LIN {X 0,Y 122.417,Z 271.708,A -85,B 0,C 180,E1 -25566.608,E2 -25566.608} C_VEL
LIN {X 0,Y 122.316,Z 271.702,A -85,B 0,C 180,E1 -25572.377,E2 -25572.377} C_VEL
LIN {X 0,Y 122.102,Z 271.77,A -85,B 0,C 180,E1 -25576.74,E2 -25576.74} C_VEL
LIN {X 0,Y 122.036,Z 271.748,A -85,B 0,C 180,E1 -25582.868,E2 -25582.868} C_VEL
LIN {X 0,Y 121.951,Z 271.777,A -85,B 0,C 180,E1 -25587.47,E2 -25587.47} C_VEL
LIN {X 0,Y 121.974,Z 272.027,A -85,B 0,C 180,E1 -25592.04,E2 -25592.04} C_VEL
LIN {X 0,Y 122.267,Z 273.161,A -85,B 0,C 180,E1 -25592.746,E2 -25592.746} C_VEL
LIN {X 0,Y 123.853,Z 275.808,A -85,B 0,C 180,E1 -25593.851,E2 -25593.851} C_VEL
LIN {X 0,Y 125.36,Z 277.295,A -85,B 0,C 180,E1 -25594.741,E2 -25594.741} C_VEL
LIN {X 0,Y 127.561,Z 280.725,A -85,B 0,C 180,E1 -25596.09,E2 -25596.09} C_VEL
LIN {X 0,Y 133.318,Z 289.437,A -85,B 0,C 180,E1 -25599.257,E2 -25599.257} C_VEL
LIN {X 0,Y 139.122,Z 299.64,A -85,B 0,C 180,E1 -25602.154,E2 -25602.154} C_VEL
LIN {X 0,Y 143.343,Z 310.259,A -85,B 0,C 180,E1 -25604.257,E2 -25604.257} C_VEL
LIN {X 0,Y 147.015,Z 321.622,A -85,B 0,C 180,E1 -25606.074,E2 -25606.074} C_VEL
LIN {X 0,Y 147.266,Z 325.906,A -85,B 0,C 180,E1 -25606.408,E2 -25606.408} C_VEL
LIN {X 0,Y 144.065,Z 374.094,A -85,B 0,C 180,E1 -25608.57,E2 -25608.57} C_VEL
LIN {X 0,Y 142.298,Z 387.376,A -85,B 0,C 180,E1 -25609.638,E2 -25609.638} C_VEL
LIN {X 0,Y 140.096,Z 399.712,A -85,B 0,C 180,E1 -25611.167,E2 -25611.167} C_VEL
LIN {X 0,Y 137.398,Z 410.903,A -85,B 0,C 180,E1 -25613.058,E2 -25613.058} C_VEL
LIN {X 0,Y 134.822,Z 419.925,A -85,B 0,C 180,E1 -25615.013,E2 -25615.013} C_VEL
LIN {X 0,Y 131.525,Z 430.91,A -85,B 0,C 180,E1 -25618.154,E2 -25618.154} C_VEL
LIN {X 0,Y 128.19,Z 440.642,A -85,B 0,C 180,E1 -25621.736,E2 -25621.736} C_VEL
LIN {X 0,Y 125.67,Z 448.029,A -85,B 0,C 180,E1 -25625.203,E2 -25625.203} C_VEL
LIN {X 0,Y 122.916,Z 456.04,A -85,B 0,C 180,E1 -25629.938,E2 -25629.938} C_VEL
LIN {X 0,Y 121.019,Z 462.413,A -85,B 0,C 180,E1 -25634.852,E2 -25634.852} C_VEL
LIN {X 0,Y 119.82,Z 467.456,A -85,B 0,C 180,E1 -25639.866,E2 -25639.866} C_VEL
LIN {X 0,Y 119.27,Z 471.332,A -85,B 0,C 180,E1 -25644.93,E2 -25644.93} C_VEL
LIN {X 0,Y 119.304,Z 474.157,A -85,B 0,C 180,E1 -25650.001,E2 -25650.001} C_VEL
LIN {X 0,Y 119.247,Z 475.469,A -85,B 0,C 180,E1 -25653.38,E2 -25653.38} C_VEL
LIN {X 0,Y 119.98,Z 476.932,A -85,B 0,C 180,E1 -25660.122,E2 -25660.122} C_VEL
LIN {X 0,Y 121.968,Z 476.809,A -85,B 0,C 180,E1 -25666.691,E2 -25666.691} C_VEL
LIN {X 0,Y 125.493,Z 475.157,A -85,B 0,C 180,E1 -25673.081,E2 -25673.081} C_VEL
LIN {X 0,Y 127.894,Z 473.752,A -85,B 0,C 180,E1 -25676.08,E2 -25676.08} C_VEL
LIN {X 0,Y 131.395,Z 471.343,A -85,B 0,C 180,E1 -25679.691,E2 -25679.691} C_VEL
LIN {X 0,Y 133.223,Z 469.569,A -85,B 0,C 180,E1 -25682.001,E2 -25682.001} C_VEL
LIN {X 0,Y 134.965,Z 466.294,A -85,B 0,C 180,E1 -25685.937,E2 -25685.937} C_VEL
LIN {X 0,Y 137.186,Z 462.408,A -85,B 0,C 180,E1 -25689.659,E2 -25689.659} C_VEL
LIN {X 0,Y 139.665,Z 459.633,A -85,B 0,C 180,E1 -25691.56,E2 -25691.56} C_VEL
LIN {X 0,Y 146.623,Z 452.507,A -85,B 0,C 180,E1 -25694.993,E2 -25694.993} C_VEL
LIN {X 0,Y 153.812,Z 443.935,A -85,B 0,C 180,E1 -25697.946,E2 -25697.946} C_VEL
LIN {X 0,Y 160.067,Z 435.206,A -85,B 0,C 180,E1 -25700.208,E2 -25700.208} C_VEL
LIN {X 0,Y 165.907,Z 425.657,A -85,B 0,C 180,E1 -25702.091,E2 -25702.091} C_VEL
LIN {X 0,Y 171.308,Z 415.227,A -85,B 0,C 180,E1 -25703.624,E2 -25703.624} C_VEL
LIN {X 0,Y 176.137,Z 403.695,A -85,B 0,C 180,E1 -25704.883,E2 -25704.883} C_VEL
LIN {X 0,Y 180.007,Z 391.632,A -85,B 0,C 180,E1 -25705.852,E2 -25705.852} C_VEL
LIN {X 0,Y 183.062,Z 378.393,A -85,B 0,C 180,E1 -25706.585,E2 -25706.585} C_VEL
LIN {X 0,Y 184.796,Z 365.742,A -85,B 0,C 180,E1 -25707.042,E2 -25707.042} C_VEL
LIN {X 0,Y 185.317,Z 359.615,A -85,B 0,C 180,E1 -25707.264,E2 -25707.264} C_VEL
LIN {X 0,Y 182.402,Z 351.71,A -85,B 0,C 180,E1 -25710.159,E2 -25710.159} C_VEL
LIN {X 0,Y 179.342,Z 344.498,A -85,B 0,C 180,E1 -25713.644,E2 -25713.644} C_VEL
LIN {X 0,Y 177.139,Z 339.924,A -85,B 0,C 180,E1 -25716.615,E2 -25716.615} C_VEL
LIN {X 0,Y 175.755,Z 337.207,A -85,B 0,C 180,E1 -25718.897,E2 -25718.897} C_VEL
LIN {X 0,Y 173.712,Z 333.275,A -85,B 0,C 180,E1 -25723.538,E2 -25723.538} C_VEL
LIN {X 0,Y 172.304,Z 331.593,A -85,B 0,C 180,E1 -25730.6,E2 -25730.6} C_VEL
LIN {X 0,Y 173.403,Z 332.544,A -85,B 0,C 180,E1 -25737.667,E2 -25737.667} C_VEL
LIN {X 0,Y 173.905,Z 333.209,A -85,B 0,C 180,E1 -25739.121,E2 -25739.121} C_VEL
LIN {X 0,Y 175.898,Z 336.978,A -85,B 0,C 180,E1 -25743.5,E2 -25743.5} C_VEL
LIN {X 0,Y 178.522,Z 341.814,A -85,B 0,C 180,E1 -25747.418,E2 -25747.418} C_VEL
LIN {X 0,Y 180.756,Z 345.931,A -85,B 0,C 180,E1 -25750.065,E2 -25750.065} C_VEL
LIN {X 0,Y 182.611,Z 349.737,A -85,B 0,C 180,E1 -25752.028,E2 -25752.028} C_VEL
LIN {X 0,Y 185.533,Z 357.045,A -85,B 0,C 180,E1 -25754.874,E2 -25754.874} C_VEL
LIN {X 0,Y 183.565,Z 374.418,A -85,B 0,C 180,E1 -25755.499,E2 -25755.499} C_VEL
LIN {X 0,Y 180.942,Z 386.69,A -85,B 0,C 180,E1 -25756.119,E2 -25756.119} C_VEL
LIN {X 0,Y 177.256,Z 398.948,A -85,B 0,C 180,E1 -25757.071,E2 -25757.071} C_VEL
LIN {X 0,Y 172.252,Z 411.617,A -85,B 0,C 180,E1 -25758.446,E2 -25758.446} C_VEL
LIN {X 0,Y 167.111,Z 421.976,A -85,B 0,C 180,E1 -25759.962,E2 -25759.962} C_VEL
LIN {X 0,Y 160.993,Z 432.133,A -85,B 0,C 180,E1 -25761.927,E2 -25761.927} C_VEL
LIN {X 0,Y 154.339,Z 441.539,A -85,B 0,C 180,E1 -25764.393,E2 -25764.393} C_VEL
LIN {X 0,Y 148,Z 449.237,A -85,B 0,C 180,E1 -25767.078,E2 -25767.078} C_VEL
LIN {X 0,Y 141.389,Z 456.166,A -85,B 0,C 180,E1 -25770.301,E2 -25770.301} C_VEL
LIN {X 0,Y 135.346,Z 461.683,A -85,B 0,C 180,E1 -25773.816,E2 -25773.816} C_VEL
LIN {X 0,Y 129.352,Z 466.403,A -85,B 0,C 180,E1 -25778.016,E2 -25778.016} C_VEL
LIN {X 0,Y 123.843,Z 470.088,A -85,B 0,C 180,E1 -25782.899,E2 -25782.899} C_VEL
LIN {X 0,Y 121.135,Z 471.63,A -85,B 0,C 180,E1 -25785.874,E2 -25785.874} C_VEL
LIN {X 0,Y 117.41,Z 473.328,A -85,B 0,C 180,E1 -25791.065,E2 -25791.065} C_VEL
LIN {X 0,Y 114.591,Z 474.002,A -85,B 0,C 180,E1 -25796.496,E2 -25796.496} C_VEL
LIN {X 0,Y 113.253,Z 473.913,A -85,B 0,C 180,E1 -25800.281,E2 -25800.281} C_VEL
LIN {X 0,Y 112.337,Z 473.353,A -85,B 0,C 180,E1 -25804.027,E2 -25804.027} C_VEL
LIN {X 0,Y 111.648,Z 471.307,A -85,B 0,C 180,E1 -25810.716,E2 -25810.716} C_VEL
LIN {X 0,Y 111.953,Z 467.915,A -85,B 0,C 180,E1 -25817.306,E2 -25817.306} C_VEL
LIN {X 0,Y 113.091,Z 463.049,A -85,B 0,C 180,E1 -25823.712,E2 -25823.712} C_VEL
LIN {X 0,Y 115.123,Z 456.472,A -85,B 0,C 180,E1 -25829.999,E2 -25829.999} C_VEL
LIN {X 0,Y 117.55,Z 449.355,A -85,B 0,C 180,E1 -25835.144,E2 -25835.144} C_VEL
LIN {X 0,Y 120.797,Z 440.409,A -85,B 0,C 180,E1 -25840.051,E2 -25840.051} C_VEL
LIN {X 0,Y 124.177,Z 431.212,A -85,B 0,C 180,E1 -25843.917,E2 -25843.917} C_VEL
LIN {X 0,Y 127.578,Z 421.06,A -85,B 0,C 180,E1 -25847.222,E2 -25847.222} C_VEL
LIN {X 0,Y 130.961,Z 409.719,A -85,B 0,C 180,E1 -25850.004,E2 -25850.004} C_VEL
LIN {X 0,Y 134.071,Z 397.023,A -85,B 0,C 180,E1 -25852.335,E2 -25852.335} C_VEL
LIN {X 0,Y 136.353,Z 384.7,A -85,B 0,C 180,E1 -25853.946,E2 -25853.946} C_VEL
LIN {X 0,Y 138.276,Z 370.597,A -85,B 0,C 180,E1 -25855.122,E2 -25855.122} C_VEL
LIN {X 0,Y 141.666,Z 320.771,A -85,B 0,C 180,E1 -25857.421,E2 -25857.421} C_VEL
LIN {X 0,Y 138.482,Z 311.486,A -85,B 0,C 180,E1 -25859.089,E2 -25859.089} C_VEL
LIN {X 0,Y 131.285,Z 297.708,A -85,B 0,C 180,E1 -25862.78,E2 -25862.78} C_VEL
LIN {X 0,Y 124.325,Z 286.522,A -85,B 0,C 180,E1 -25866.815,E2 -25866.815} C_VEL
LIN {X 0,Y 121.077,Z 282.094,A -85,B 0,C 180,E1 -25868.889,E2 -25868.889} C_VEL
LIN {X 0,Y 118.948,Z 279.166,A -85,B 0,C 180,E1 -25870.362,E2 -25870.362} C_VEL
LIN {X 0,Y 118.239,Z 277.828,A -85,B 0,C 180,E1 -25870.91,E2 -25870.91} C_VEL
LIN {X 0,Y 115.881,Z 275.514,A -85,B 0,C 180,E1 -25872.61,E2 -25872.61} C_VEL
LIN {X 0,Y 114.976,Z 273.193,A -85,B 0,C 180,E1 -25873.766,E2 -25873.766} C_VEL
LIN {X 0,Y 114.847,Z 272.682,A -85,B 0,C 180,E1 -25875.203,E2 -25875.203} C_VEL
LIN {X 0,Y 114.852,Z 272.662,A -85,B 0,C 180,E1 -25877.716,E2 -25877.716} C_VEL
LIN {X 0,Y 114.833,Z 272.637,A -85,B 0,C 180,E1 -25882.712,E2 -25882.712} C_VEL
LIN {X 0,Y 114.844,Z 272.645,A -85,B 0,C 180,E1 -25888.95,E2 -25888.95} C_VEL
LIN {X 0,Y 114.946,Z 272.645,A -85,B 0,C 180,E1 -25896.506,E2 -25896.506} C_VEL
LIN {X 0,Y 115.016,Z 272.604,A -85,B 0,C 180,E1 -25902.228,E2 -25902.228} C_VEL
LIN {X 0,Y 115.276,Z 272.57,A -85,B 0,C 180,E1 -25907.276,E2 -25907.276} C_VEL
LIN {X 0,Y 115.387,Z 272.593,A -85,B 0,C 180,E1 -25913.019,E2 -25913.019} C_VEL
LIN {X 0,Y 115.989,Z 272.479,A -85,B 0,C 180,E1 -25920.016,E2 -25920.016} C_VEL
LIN {X 0,Y 115.359,Z 272.578,A -85,B 0,C 180,E1 -25927.014,E2 -25927.014} C_VEL
LIN {X 0,Y 115.252,Z 272.583,A -85,B 0,C 180,E1 -25932.672,E2 -25932.672} C_VEL
LIN {X 0,Y 115.006,Z 272.635,A -85,B 0,C 180,E1 -25937.807,E2 -25937.807} C_VEL
LIN {X 0,Y 114.955,Z 272.635,A -85,B 0,C 180,E1 -25943.505,E2 -25943.505} C_VEL
LIN {X 0,Y 114.957,Z 272.956,A -85,B 0,C 180,E1 -25947.802,E2 -25947.802} C_VEL
LIN {X 0,Y 115.218,Z 274.115,A -85,B 0,C 180,E1 -25948.6,E2 -25948.6} C_VEL
LIN {X 0,Y 116.721,Z 276.593,A -85,B 0,C 180,E1 -25949.868,E2 -25949.868} C_VEL
LIN {X 0,Y 118.61,Z 278.382,A -85,B 0,C 180,E1 -25951.197,E2 -25951.197} C_VEL
LIN {X 0,Y 120.6,Z 281.579,A -85,B 0,C 180,E1 -25952.635,E2 -25952.635} C_VEL
LIN {X 0,Y 122.018,Z 283.329,A -85,B 0,C 180,E1 -25953.56,E2 -25953.56} C_VEL
LIN {X 0,Y 127.424,Z 291.559,A -85,B 0,C 180,E1 -25956.909,E2 -25956.909} C_VEL
LIN {X 0,Y 132.932,Z 300.828,A -85,B 0,C 180,E1 -25959.946,E2 -25959.946} C_VEL
LIN {X 0,Y 135.86,Z 307.143,A -85,B 0,C 180,E1 -25961.513,E2 -25961.513} C_VEL
LIN {X 0,Y 140.144,Z 319.557,A -85,B 0,C 180,E1 -25963.842,E2 -25963.842} C_VEL
LIN {X 0,Y 141.499,Z 323.985,A -85,B 0,C 180,E1 -25964.567,E2 -25964.567} C_VEL
LIN {X 0,Y 141.281,Z 330.164,A -85,B 0,C 180,E1 -25964.901,E2 -25964.901} C_VEL
LIN {X 0,Y 138.295,Z 373.676,A -85,B 0,C 180,E1 -25966.913,E2 -25966.913} C_VEL
LIN {X 0,Y 136.449,Z 386.809,A -85,B 0,C 180,E1 -25967.967,E2 -25967.967} C_VEL
LIN {X 0,Y 134.122,Z 399.503,A -85,B 0,C 180,E1 -25969.577,E2 -25969.577} C_VEL
LIN {X 0,Y 131.296,Z 410.723,A -85,B 0,C 180,E1 -25971.52,E2 -25971.52} C_VEL
LIN {X 0,Y 128.599,Z 419.757,A -85,B 0,C 180,E1 -25973.537,E2 -25973.537} C_VEL
LIN {X 0,Y 125.121,Z 430.755,A -85,B 0,C 180,E1 -25976.795,E2 -25976.795} C_VEL
LIN {X 0,Y 121.982,Z 439.354,A -85,B 0,C 180,E1 -25980.033,E2 -25980.033} C_VEL
LIN {X 0,Y 119.227,Z 447.141,A -85,B 0,C 180,E1 -25983.764,E2 -25983.764} C_VEL
LIN {X 0,Y 116.255,Z 455.298,A -85,B 0,C 180,E1 -25988.734,E2 -25988.734} C_VEL
LIN {X 0,Y 114.127,Z 461.826,A -85,B 0,C 180,E1 -25993.913,E2 -25993.913} C_VEL
LIN {X 0,Y 112.811,Z 466.979,A -85,B 0,C 180,E1 -25999.23,E2 -25999.23} C_VEL
LIN {X 0,Y 112.211,Z 470.953,A -85,B 0,C 180,E1 -26004.61,E2 -26004.61} C_VEL
LIN {X 0,Y 112.224,Z 473.863,A -85,B 0,C 180,E1 -26010.001,E2 -26010.001} C_VEL
LIN {X 0,Y 112.158,Z 475.222,A -85,B 0,C 180,E1 -26013.594,E2 -26013.594} C_VEL
LIN {X 0,Y 112.979,Z 476.77,A -85,B 0,C 180,E1 -26020.757,E2 -26020.757} C_VEL
LIN {X 0,Y 113.875,Z 476.975,A -85,B 0,C 180,E1 -26024.293,E2 -26024.293} C_VEL
LIN {X 0,Y 116.866,Z 476.175,A -85,B 0,C 180,E1 -26031.152,E2 -26031.152} C_VEL
LIN {X 0,Y 121.555,Z 473.854,A -85,B 0,C 180,E1 -26037.552,E2 -26037.552} C_VEL
LIN {X 0,Y 126.015,Z 471.017,A -85,B 0,C 180,E1 -26041.995,E2 -26041.995} C_VEL
LIN {X 0,Y 131.173,Z 467.188,A -85,B 0,C 180,E1 -26046.113,E2 -26046.113} C_VEL
LIN {X 0,Y 136.846,Z 462.277,A -85,B 0,C 180,E1 -26049.939,E2 -26049.939} C_VEL
LIN {X 0,Y 139.665,Z 459.633,A -85,B 0,C 180,E1 -26051.56,E2 -26051.56} C_VEL
LIN {X 0,Y 142.267,Z 456.671,A -85,B 0,C 180,E1 -26053.355,E2 -26053.355} C_VEL
LIN {X 0,Y 145.332,Z 451.535,A -85,B 0,C 180,E1 -26056.516,E2 -26056.516} C_VEL
LIN {X 0,Y 148.596,Z 445.868,A -85,B 0,C 180,E1 -26059.403,E2 -26059.403} C_VEL
LIN {X 0,Y 151.391,Z 441.999,A -85,B 0,C 180,E1 -26060.736,E2 -26060.736} C_VEL
LIN {X 0,Y 158.282,Z 432.309,A -85,B 0,C 180,E1 -26063.058,E2 -26063.058} C_VEL
LIN {X 0,Y 164.465,Z 422.062,A -85,B 0,C 180,E1 -26064.812,E2 -26064.812} C_VEL
LIN {X 0,Y 170.07,Z 410.735,A -85,B 0,C 180,E1 -26066.269,E2 -26066.269} C_VEL
LIN {X 0,Y 174.697,Z 398.947,A -85,B 0,C 180,E1 -26067.386,E2 -26067.386} C_VEL
LIN {X 0,Y 178.488,Z 385.83,A -85,B 0,C 180,E1 -26068.269,E2 -26068.269} C_VEL
LIN {X 0,Y 181.136,Z 372.198,A -85,B 0,C 180,E1 -26068.873,E2 -26068.873} C_VEL
LIN {X 0,Y 182.137,Z 362.932,A -85,B 0,C 180,E1 -26069.188,E2 -26069.188} C_VEL
LIN {X 0,Y 179.796,Z 356.395,A -85,B 0,C 180,E1 -26071.778,E2 -26071.778} C_VEL
LIN {X 0,Y 177.285,Z 350.146,A -85,B 0,C 180,E1 -26074.957,E2 -26074.957} C_VEL
LIN {X 0,Y 175.505,Z 346.105,A -85,B 0,C 180,E1 -26077.63,E2 -26077.63} C_VEL
LIN {X 0,Y 174.398,Z 343.857,A -85,B 0,C 180,E1 -26079.651,E2 -26079.651} C_VEL
LIN {X 0,Y 172.635,Z 340.214,A -85,B 0,C 180,E1 -26084.011,E2 -26084.011} C_VEL
LIN {X 0,Y 171.414,Z 338.641,A -85,B 0,C 180,E1 -26090.551,E2 -26090.551} C_VEL
LIN {X 0,Y 172.232,Z 339.43,A -85,B 0,C 180,E1 -26096.802,E2 -26096.802} C_VEL
LIN {X 0,Y 172.806,Z 340.031,A -85,B 0,C 180,E1 -26098.591,E2 -26098.591} C_VEL
LIN {X 0,Y 174.975,Z 344.508,A -85,B 0,C 180,E1 -26103.578,E2 -26103.578} C_VEL
LIN {X 0,Y 177.144,Z 348.707,A -85,B 0,C 180,E1 -26106.927,E2 -26106.927} C_VEL
LIN {X 0,Y 179.642,Z 353.549,A -85,B 0,C 180,E1 -26109.986,E2 -26109.986} C_VEL
LIN {X 0,Y 182.359,Z 360.523,A -85,B 0,C 180,E1 -26112.964,E2 -26112.964} C_VEL
LIN {X 0,Y 180.474,Z 375.476,A -85,B 0,C 180,E1 -26113.501,E2 -26113.501} C_VEL
LIN {X 0,Y 177.5,Z 388.399,A -85,B 0,C 180,E1 -26114.177,E2 -26114.177} C_VEL
LIN {X 0,Y 173.403,Z 401.121,A -85,B 0,C 180,E1 -26115.177,E2 -26115.177} C_VEL
LIN {X 0,Y 168.534,Z 412.688,A -85,B 0,C 180,E1 -26116.438,E2 -26116.438} C_VEL
LIN {X 0,Y 162.652,Z 423.802,A -85,B 0,C 180,E1 -26118.084,E2 -26118.084} C_VEL
LIN {X 0,Y 156.209,Z 433.882,A -85,B 0,C 180,E1 -26120.082,E2 -26120.082} C_VEL
LIN {X 0,Y 149.656,Z 442.606,A -85,B 0,C 180,E1 -26122.422,E2 -26122.422} C_VEL
LIN {X 0,Y 142.125,Z 451.07,A -85,B 0,C 180,E1 -26125.516,E2 -26125.516} C_VEL
LIN {X 0,Y 134.719,Z 458.136,A -85,B 0,C 180,E1 -26129.094,E2 -26129.094} C_VEL
LIN {X 0,Y 127.358,Z 464.145,A -85,B 0,C 180,E1 -26133.474,E2 -26133.474} C_VEL
LIN {X 0,Y 120.903,Z 468.547,A -85,B 0,C 180,E1 -26138.301,E2 -26138.301} C_VEL
LIN {X 0,Y 115.753,Z 471.446,A -85,B 0,C 180,E1 -26143.231,E2 -26143.231} C_VEL
LIN {X 0,Y 111.026,Z 473.455,A -85,B 0,C 180,E1 -26149.401,E2 -26149.401} C_VEL
LIN {X 0,Y 108.294,Z 474.075,A -85,B 0,C 180,E1 -26154.261,E2 -26154.261} C_VEL
LIN {X 0,Y 106.434,Z 474.007,A -85,B 0,C 180,E1 -26159.101,E2 -26159.101} C_VEL
LIN {X 0,Y 104.845,Z 472.676,A -85,B 0,C 180,E1 -26166.283,E2 -26166.283} C_VEL
LIN {X 0,Y 104.566,Z 471.314,A -85,B 0,C 180,E1 -26170.362,E2 -26170.362} C_VEL
LIN {X 0,Y 104.729,Z 468.428,A -85,B 0,C 180,E1 -26176.415,E2 -26176.415} C_VEL
LIN {X 0,Y 105.605,Z 464.468,A -85,B 0,C 180,E1 -26182.35,E2 -26182.35} C_VEL
LIN {X 0,Y 107.16,Z 459.343,A -85,B 0,C 180,E1 -26188.12,E2 -26188.12} C_VEL
LIN {X 0,Y 109.452,Z 452.902,A -85,B 0,C 180,E1 -26193.68,E2 -26193.68} C_VEL
LIN {X 0,Y 112.516,Z 444.821,A -85,B 0,C 180,E1 -26198.983,E2 -26198.983} C_VEL
LIN {X 0,Y 115.686,Z 436.573,A -85,B 0,C 180,E1 -26203.168,E2 -26203.168} C_VEL
LIN {X 0,Y 119.074,Z 427.569,A -85,B 0,C 180,E1 -26206.721,E2 -26206.721} C_VEL
LIN {X 0,Y 122.885,Z 416.492,A -85,B 0,C 180,E1 -26210.068,E2 -26210.068} C_VEL
LIN {X 0,Y 126.086,Z 405.614,A -85,B 0,C 180,E1 -26212.531,E2 -26212.531} C_VEL
LIN {X 0,Y 129.083,Z 392.588,A -85,B 0,C 180,E1 -26214.742,E2 -26214.742} C_VEL
LIN {X 0,Y 131.437,Z 379.529,A -85,B 0,C 180,E1 -26216.227,E2 -26216.227} C_VEL
LIN {X 0,Y 133.028,Z 365.638,A -85,B 0,C 180,E1 -26217.197,E2 -26217.197} C_VEL
LIN {X 0,Y 136.059,Z 322.609,A -85,B 0,C 180,E1 -26219.163,E2 -26219.163} C_VEL
LIN {X 0,Y 133.508,Z 315.096,A -85,B 0,C 180,E1 -26220.622,E2 -26220.622} C_VEL
LIN {X 0,Y 127.034,Z 302.351,A -85,B 0,C 180,E1 -26224.232,E2 -26224.232} C_VEL
LIN {X 0,Y 120.806,Z 292.065,A -85,B 0,C 180,E1 -26228.131,E2 -26228.131} C_VEL
LIN {X 0,Y 117.403,Z 287.353,A -85,B 0,C 180,E1 -26230.48,E2 -26230.48} C_VEL
LIN {X 0,Y 114.772,Z 283.47,A -85,B 0,C 180,E1 -26232.507,E2 -26232.507} C_VEL
LIN {X 0,Y 112.455,Z 280.581,A -85,B 0,C 180,E1 -26234.399,E2 -26234.399} C_VEL
LIN {X 0,Y 111.521,Z 278.954,A -85,B 0,C 180,E1 -26235.262,E2 -26235.262} C_VEL
LIN {X 0,Y 109.242,Z 277.027,A -85,B 0,C 180,E1 -26237.253,E2 -26237.253} C_VEL
LIN {X 0,Y 107.83,Z 274.109,A -85,B 0,C 180,E1 -26239.154,E2 -26239.154} C_VEL
LIN {X 0,Y 107.716,Z 273.577,A -85,B 0,C 180,E1 -26240.565,E2 -26240.565} C_VEL
LIN {X 0,Y 107.743,Z 273.53,A -85,B 0,C 180,E1 -26244.074,E2 -26244.074} C_VEL
LIN {X 0,Y 107.786,Z 273.527,A -85,B 0,C 180,E1 -26248.58,E2 -26248.58} C_VEL
LIN {X 0,Y 107.911,Z 273.527,A -85,B 0,C 180,E1 -26257.017,E2 -26257.017} C_VEL
LIN {X 0,Y 108.032,Z 273.458,A -85,B 0,C 180,E1 -26264.935,E2 -26264.935} C_VEL
LIN {X 0,Y 108.282,Z 273.459,A -85,B 0,C 180,E1 -26268.79,E2 -26268.79} C_VEL
LIN {X 0,Y 108.452,Z 273.411,A -85,B 0,C 180,E1 -26276.301,E2 -26276.301} C_VEL
LIN {X 0,Y 108.915,Z 273.359,A -85,B 0,C 180,E1 -26280.017,E2 -26280.017} C_VEL
LIN {X 0,Y 108.299,Z 273.45,A -85,B 0,C 180,E1 -26287.474,E2 -26287.474} C_VEL
LIN {X 0,Y 108.174,Z 273.466,A -85,B 0,C 180,E1 -26292.963,E2 -26292.963} C_VEL
LIN {X 0,Y 107.93,Z 273.587,A -85,B 0,C 180,E1 -26302.005,E2 -26302.005} C_VEL
LIN {X 0,Y 108.139,Z 274.54,A -85,B 0,C 180,E1 -26303.263,E2 -26303.263} C_VEL
LIN {X 0,Y 109.443,Z 277.213,A -85,B 0,C 180,E1 -26304.766,E2 -26304.766} C_VEL
LIN {X 0,Y 111.856,Z 279.375,A -85,B 0,C 180,E1 -26306.863,E2 -26306.863} C_VEL
LIN {X 0,Y 113.834,Z 282.544,A -85,B 0,C 180,E1 -26308.603,E2 -26308.603} C_VEL
LIN {X 0,Y 115.53,Z 284.462,A -85,B 0,C 180,E1 -26309.914,E2 -26309.914} C_VEL
LIN {X 0,Y 118.058,Z 288.055,A -85,B 0,C 180,E1 -26311.804,E2 -26311.804} C_VEL
LIN {X 0,Y 123.538,Z 296.63,A -85,B 0,C 180,E1 -26315.492,E2 -26315.492} C_VEL
LIN {X 0,Y 128.718,Z 305.709,A -85,B 0,C 180,E1 -26318.598,E2 -26318.598} C_VEL
LIN {X 0,Y 131.317,Z 311.694,A -85,B 0,C 180,E1 -26320.115,E2 -26320.115} C_VEL
LIN {X 0,Y 134.971,Z 322.649,A -85,B 0,C 180,E1 -26322.287,E2 -26322.287} C_VEL
LIN {X 0,Y 135.988,Z 326.269,A -85,B 0,C 180,E1 -26322.899,E2 -26322.899} C_VEL
LIN {X 0,Y 132.585,Z 373.615,A -85,B 0,C 180,E1 -26325.131,E2 -26325.131} C_VEL
LIN {X 0,Y 130.705,Z 386.557,A -85,B 0,C 180,E1 -26326.19,E2 -26326.19} C_VEL
LIN {X 0,Y 128.262,Z 399.293,A -85,B 0,C 180,E1 -26327.84,E2 -26327.84} C_VEL
LIN {X 0,Y 125.296,Z 410.542,A -85,B 0,C 180,E1 -26329.832,E2 -26329.832} C_VEL
LIN {X 0,Y 122.468,Z 419.588,A -85,B 0,C 180,E1 -26331.911,E2 -26331.911} C_VEL
LIN {X 0,Y 118.795,Z 430.602,A -85,B 0,C 180,E1 -26335.292,E2 -26335.292} C_VEL
LIN {X 0,Y 114.937,Z 440.733,A -85,B 0,C 180,E1 -26339.361,E2 -26339.361} C_VEL
LIN {X 0,Y 112.245,Z 447.756,A -85,B 0,C 180,E1 -26343.004,E2 -26343.004} C_VEL
LIN {X 0,Y 109.148,Z 455.783,A -85,B 0,C 180,E1 -26348.271,E2 -26348.271} C_VEL
LIN {X 0,Y 107.288,Z 461.201,A -85,B 0,C 180,E1 -26352.857,E2 -26352.857} C_VEL
LIN {X 0,Y 105.832,Z 466.48,A -85,B 0,C 180,E1 -26358.51,E2 -26358.51} C_VEL
LIN {X 0,Y 105.13,Z 470.55,A -85,B 0,C 180,E1 -26364.246,E2 -26364.246} C_VEL
LIN {X 0,Y 105.131,Z 473.538,A -85,B 0,C 180,E1 -26370.001,E2 -26370.001} C_VEL
LIN {X 0,Y 105.093,Z 474.976,A -85,B 0,C 180,E1 -26373.836,E2 -26373.836} C_VEL
LIN {X 0,Y 106.005,Z 476.607,A -85,B 0,C 180,E1 -26381.474,E2 -26381.474} C_VEL
LIN {X 0,Y 108.444,Z 476.727,A -85,B 0,C 180,E1 -26388.909,E2 -26388.909} C_VEL
LIN {X 0,Y 112.564,Z 475.255,A -85,B 0,C 180,E1 -26395.917,E2 -26395.917} C_VEL
LIN {X 0,Y 118.383,Z 472.244,A -85,B 0,C 180,E1 -26402.297,E2 -26402.297} C_VEL
LIN {X 0,Y 123.627,Z 468.842,A -85,B 0,C 180,E1 -26406.65,E2 -26406.65} C_VEL
LIN {X 0,Y 129.41,Z 464.406,A -85,B 0,C 180,E1 -26410.671,E2 -26410.671} C_VEL
LIN {X 0,Y 137.018,Z 457.736,A -85,B 0,C 180,E1 -26414.853,E2 -26414.853} C_VEL
LIN {X 0,Y 144.179,Z 450.492,A -85,B 0,C 180,E1 -26418.02,E2 -26418.02} C_VEL
LIN {X 0,Y 151.391,Z 441.999,A -85,B 0,C 180,E1 -26420.736,E2 -26420.736} C_VEL
LIN {X 0,Y 154.168,Z 437.992,A -85,B 0,C 180,E1 -26421.993,E2 -26421.993} C_VEL
LIN {X 0,Y 157.434,Z 431.271,A -85,B 0,C 180,E1 -26424.4,E2 -26424.4} C_VEL
LIN {X 0,Y 160.495,Z 424.042,A -85,B 0,C 180,E1 -26426.575,E2 -26426.575} C_VEL
LIN {X 0,Y 162.838,Z 419.246,A -85,B 0,C 180,E1 -26427.458,E2 -26427.458} C_VEL
LIN {X 0,Y 168.476,Z 407.536,A -85,B 0,C 180,E1 -26428.779,E2 -26428.779} C_VEL
LIN {X 0,Y 173.241,Z 394.689,A -85,B 0,C 180,E1 -26429.847,E2 -26429.847} C_VEL
LIN {X 0,Y 176.633,Z 382.131,A -85,B 0,C 180,E1 -26430.558,E2 -26430.558} C_VEL
LIN {X 0,Y 178.947,Z 368.334,A -85,B 0,C 180,E1 -26431.091,E2 -26431.091} C_VEL
LIN {X 0,Y 179.167,Z 366.343,A -85,B 0,C 180,E1 -26431.169,E2 -26431.169} C_VEL
LIN {X 0,Y 176.927,Z 359.883,A -85,B 0,C 180,E1 -26434.001,E2 -26434.001} C_VEL
LIN {X 0,Y 175.248,Z 355.597,A -85,B 0,C 180,E1 -26436.418,E2 -26436.418} C_VEL
LIN {X 0,Y 173.878,Z 352.113,A -85,B 0,C 180,E1 -26438.813,E2 -26438.813} C_VEL
LIN {X 0,Y 173.003,Z 350.38,A -85,B 0,C 180,E1 -26440.563,E2 -26440.563} C_VEL
LIN {X 0,Y 171.552,Z 347.122,A -85,B 0,C 180,E1 -26444.546,E2 -26444.546} C_VEL
LIN {X 0,Y 170.525,Z 345.679,A -85,B 0,C 180,E1 -26450.501,E2 -26450.501} C_VEL
LIN {X 0,Y 171.329,Z 346.478,A -85,B 0,C 180,E1 -26456.785,E2 -26456.785} C_VEL
LIN {X 0,Y 171.746,Z 347.02,A -85,B 0,C 180,E1 -26458.172,E2 -26458.172} C_VEL
LIN {X 0,Y 173.647,Z 351.189,A -85,B 0,C 180,E1 -26462.889,E2 -26462.889} C_VEL
LIN {X 0,Y 175.648,Z 355.366,A -85,B 0,C 180,E1 -26466.245,E2 -26466.245} C_VEL
LIN {X 0,Y 177.767,Z 359.748,A -85,B 0,C 180,E1 -26469.031,E2 -26469.031} C_VEL
LIN {X 0,Y 179.378,Z 364.052,A -85,B 0,C 180,E1 -26470.982,E2 -26470.982} C_VEL
LIN {X 0,Y 177.463,Z 377.068,A -85,B 0,C 180,E1 -26471.457,E2 -26471.457} C_VEL
LIN {X 0,Y 174.439,Z 389.48,A -85,B 0,C 180,E1 -26472.111,E2 -26472.111} C_VEL
LIN {X 0,Y 170.425,Z 401.444,A -85,B 0,C 180,E1 -26473.028,E2 -26473.028} C_VEL
LIN {X 0,Y 165.307,Z 413.171,A -85,B 0,C 180,E1 -26474.279,E2 -26474.279} C_VEL
LIN {X 0,Y 158.98,Z 424.653,A -85,B 0,C 180,E1 -26475.948,E2 -26475.948} C_VEL
LIN {X 0,Y 152.326,Z 434.604,A -85,B 0,C 180,E1 -26477.899,E2 -26477.899} C_VEL
LIN {X 0,Y 145.528,Z 443.197,A -85,B 0,C 180,E1 -26480.191,E2 -26480.191} C_VEL
LIN {X 0,Y 137.69,Z 451.559,A -85,B 0,C 180,E1 -26483.253,E2 -26483.253} C_VEL
LIN {X 0,Y 129.941,Z 458.553,A -85,B 0,C 180,E1 -26486.819,E2 -26486.819} C_VEL
LIN {X 0,Y 122.405,Z 464.324,A -85,B 0,C 180,E1 -26491.095,E2 -26491.095} C_VEL
LIN {X 0,Y 116.317,Z 468.244,A -85,B 0,C 180,E1 -26495.344,E2 -26495.344} C_VEL
LIN {X 0,Y 110.648,Z 471.268,A -85,B 0,C 180,E1 -26500.34,E2 -26500.34} C_VEL
LIN {X 0,Y 107.391,Z 472.667,A -85,B 0,C 180,E1 -26503.954,E2 -26503.954} C_VEL
LIN {X 0,Y 104.585,Z 473.634,A -85,B 0,C 180,E1 -26507.778,E2 -26507.778} C_VEL
LIN {X 0,Y 102.192,Z 474.149,A -85,B 0,C 180,E1 -26511.759,E2 -26511.759} C_VEL
LIN {X 0,Y 99.651,Z 474.099,A -85,B 0,C 180,E1 -26517.775,E2 -26517.775} C_VEL
LIN {X 0,Y 97.983,Z 472.999,A -85,B 0,C 180,E1 -26524.508,E2 -26524.508} C_VEL
LIN {X 0,Y 97.493,Z 471.477,A -85,B 0,C 180,E1 -26529.516,E2 -26529.516} C_VEL
LIN {X 0,Y 97.551,Z 468.94,A -85,B 0,C 180,E1 -26535.394,E2 -26535.394} C_VEL
LIN {X 0,Y 98.341,Z 465.112,A -85,B 0,C 180,E1 -26541.781,E2 -26541.781} C_VEL
LIN {X 0,Y 99.913,Z 460.126,A -85,B 0,C 180,E1 -26547.983,E2 -26547.983} C_VEL
LIN {X 0,Y 102.247,Z 453.847,A -85,B 0,C 180,E1 -26553.94,E2 -26553.94} C_VEL
LIN {X 0,Y 105.435,Z 446.027,A -85,B 0,C 180,E1 -26559.591,E2 -26559.591} C_VEL
LIN {X 0,Y 109.095,Z 436.996,A -85,B 0,C 180,E1 -26564.508,E2 -26564.508} C_VEL
LIN {X 0,Y 113.039,Z 427.088,A -85,B 0,C 180,E1 -26568.579,E2 -26568.579} C_VEL
LIN {X 0,Y 116.62,Z 417.231,A -85,B 0,C 180,E1 -26571.66,E2 -26571.66} C_VEL
LIN {X 0,Y 119.976,Z 406.548,A -85,B 0,C 180,E1 -26574.207,E2 -26574.207} C_VEL
LIN {X 0,Y 123.132,Z 393.746,A -85,B 0,C 180,E1 -26576.481,E2 -26576.481} C_VEL
LIN {X 0,Y 125.598,Z 381.034,A -85,B 0,C 180,E1 -26578.032,E2 -26578.032} C_VEL
LIN {X 0,Y 127.356,Z 367.443,A -85,B 0,C 180,E1 -26579.046,E2 -26579.046} C_VEL
LIN {X 0,Y 130.62,Z 324.463,A -85,B 0,C 180,E1 -26581.039,E2 -26581.039} C_VEL
LIN {X 0,Y 128.718,Z 318.946,A -85,B 0,C 180,E1 -26582.216,E2 -26582.216} C_VEL
LIN {X 0,Y 122.99,Z 307.267,A -85,B 0,C 180,E1 -26585.701,E2 -26585.701} C_VEL
LIN {X 0,Y 117.131,Z 297.281,A -85,B 0,C 180,E1 -26589.681,E2 -26589.681} C_VEL
LIN {X 0,Y 111.626,Z 289.205,A -85,B 0,C 180,E1 -26594.031,E2 -26594.031} C_VEL
LIN {X 0,Y 109.028,Z 285.5,A -85,B 0,C 180,E1 -26596.4,E2 -26596.4} C_VEL
LIN {X 0,Y 106.106,Z 282.26,A -85,B 0,C 180,E1 -26599.263,E2 -26599.263} C_VEL
LIN {X 0,Y 104.948,Z 280.086,A -85,B 0,C 180,E1 -26600.637,E2 -26600.637} C_VEL
LIN {X 0,Y 102.299,Z 278.061,A -85,B 0,C 180,E1 -26603.686,E2 -26603.686} C_VEL
LIN {X 0,Y 100.822,Z 275.271,A -85,B 0,C 180,E1 -26606.13,E2 -26606.13} C_VEL
LIN {X 0,Y 100.728,Z 274.49,A -85,B 0,C 180,E1 -26607.832,E2 -26607.832} C_VEL
LIN {X 0,Y 100.77,Z 274.387,A -85,B 0,C 180,E1 -26615.284,E2 -26615.284} C_VEL
LIN {X 0,Y 100.817,Z 274.407,A -85,B 0,C 180,E1 -26619.621,E2 -26619.621} C_VEL
LIN {X 0,Y 101.18,Z 274.33,A -85,B 0,C 180,E1 -26627.991,E2 -26627.991} C_VEL
LIN {X 0,Y 101.264,Z 274.364,A -85,B 0,C 180,E1 -26632.04,E2 -26632.04} C_VEL
LIN {X 0,Y 101.842,Z 274.238,A -85,B 0,C 180,E1 -26640.018,E2 -26640.018} C_VEL
LIN {X 0,Y 101.238,Z 274.323,A -85,B 0,C 180,E1 -26647.998,E2 -26647.998} C_VEL
LIN {X 0,Y 101.037,Z 274.448,A -85,B 0,C 180,E1 -26654.24,E2 -26654.24} C_VEL
LIN {X 0,Y 101.076,Z 275.243,A -85,B 0,C 180,E1 -26656.045,E2 -26656.045} C_VEL
LIN {X 0,Y 102.413,Z 278.013,A -85,B 0,C 180,E1 -26658.264,E2 -26658.264} C_VEL
LIN {X 0,Y 104.9,Z 279.905,A -85,B 0,C 180,E1 -26661.124,E2 -26661.124} C_VEL
LIN {X 0,Y 107.307,Z 283.797,A -85,B 0,C 180,E1 -26663.82,E2 -26663.82} C_VEL
LIN {X 0,Y 109.063,Z 285.58,A -85,B 0,C 180,E1 -26665.471,E2 -26665.471} C_VEL
LIN {X 0,Y 111.486,Z 289.026,A -85,B 0,C 180,E1 -26667.682,E2 -26667.682} C_VEL
LIN {X 0,Y 115.638,Z 295.152,A -85,B 0,C 180,E1 -26671.057,E2 -26671.057} C_VEL
LIN {X 0,Y 120.961,Z 303.73,A -85,B 0,C 180,E1 -26674.822,E2 -26674.822} C_VEL
LIN {X 0,Y 125.457,Z 312.38,A -85,B 0,C 180,E1 -26677.704,E2 -26677.704} C_VEL
LIN {X 0,Y 128.593,Z 321.513,A -85,B 0,C 180,E1 -26679.763,E2 -26679.763} C_VEL
LIN {X 0,Y 130.414,Z 327.443,A -85,B 0,C 180,E1 -26680.936,E2 -26680.936} C_VEL
LIN {X 0,Y 127.041,Z 373.381,A -85,B 0,C 180,E1 -26683.179,E2 -26683.179} C_VEL
LIN {X 0,Y 124.954,Z 387.063,A -85,B 0,C 180,E1 -26684.329,E2 -26684.329} C_VEL
LIN {X 0,Y 122.523,Z 399.078,A -85,B 0,C 180,E1 -26685.935,E2 -26685.935} C_VEL
LIN {X 0,Y 119.416,Z 410.362,A -85,B 0,C 180,E1 -26687.977,E2 -26687.977} C_VEL
LIN {X 0,Y 116.448,Z 419.418,A -85,B 0,C 180,E1 -26690.116,E2 -26690.116} C_VEL
LIN {X 0,Y 112.559,Z 430.448,A -85,B 0,C 180,E1 -26693.62,E2 -26693.62} C_VEL
LIN {X 0,Y 108.41,Z 440.716,A -85,B 0,C 180,E1 -26697.924,E2 -26697.924} C_VEL
LIN {X 0,Y 105.292,Z 448.372,A -85,B 0,C 180,E1 -26702.147,E2 -26702.147} C_VEL
LIN {X 0,Y 102.568,Z 455.038,A -85,B 0,C 180,E1 -26706.798,E2 -26706.798} C_VEL
LIN {X 0,Y 100.484,Z 460.566,A -85,B 0,C 180,E1 -26711.657,E2 -26711.657} C_VEL
LIN {X 0,Y 98.851,Z 465.953,A -85,B 0,C 180,E1 -26717.686,E2 -26717.686} C_VEL
LIN {X 0,Y 98.074,Z 470.124,A -85,B 0,C 180,E1 -26723.831,E2 -26723.831} C_VEL
LIN {X 0,Y 98.032,Z 473.204,A -85,B 0,C 180,E1 -26730.001,E2 -26730.001} C_VEL
LIN {X 0,Y 98.02,Z 474.712,A -85,B 0,C 180,E1 -26734.113,E2 -26734.113} C_VEL
LIN {X 0,Y 99.036,Z 476.445,A -85,B 0,C 180,E1 -26742.293,E2 -26742.293} C_VEL
LIN {X 0,Y 101.729,Z 476.655,A -85,B 0,C 180,E1 -26750.209,E2 -26750.209} C_VEL
LIN {X 0,Y 103.699,Z 476.187,A -85,B 0,C 180,E1 -26753.995,E2 -26753.995} C_VEL
LIN {X 0,Y 109.165,Z 474.042,A -85,B 0,C 180,E1 -26761.001,E2 -26761.001} C_VEL
LIN {X 0,Y 114.201,Z 471.394,A -85,B 0,C 180,E1 -26765.779,E2 -26765.779} C_VEL
LIN {X 0,Y 119.991,Z 467.768,A -85,B 0,C 180,E1 -26770.113,E2 -26770.113} C_VEL
LIN {X 0,Y 126.319,Z 463.077,A -85,B 0,C 180,E1 -26774.065,E2 -26774.065} C_VEL
LIN {X 0,Y 134.539,Z 456.059,A -85,B 0,C 180,E1 -26778.108,E2 -26778.108} C_VEL
LIN {X 0,Y 142.143,Z 448.459,A -85,B 0,C 180,E1 -26781.146,E2 -26781.146} C_VEL
LIN {X 0,Y 150.069,Z 438.961,A -85,B 0,C 180,E1 -26783.887,E2 -26783.887} C_VEL
LIN {X 0,Y 156.965,Z 429.185,A -85,B 0,C 180,E1 -26785.928,E2 -26785.928} C_VEL
LIN {X 0,Y 162.838,Z 419.246,A -85,B 0,C 180,E1 -26787.458,E2 -26787.458} C_VEL
LIN {X 0,Y 165.107,Z 414.345,A -85,B 0,C 180,E1 -26788.269,E2 -26788.269} C_VEL
LIN {X 0,Y 167.735,Z 406.189,A -85,B 0,C 180,E1 -26790.016,E2 -26790.016} C_VEL
LIN {X 0,Y 169.918,Z 397.759,A -85,B 0,C 180,E1 -26791.617,E2 -26791.617} C_VEL
LIN {X 0,Y 171.408,Z 392.321,A -85,B 0,C 180,E1 -26792.201,E2 -26792.201} C_VEL
LIN {X 0,Y 174.818,Z 378.923,A -85,B 0,C 180,E1 -26792.877,E2 -26792.877} C_VEL
LIN {X 0,Y 176.31,Z 369.791,A -85,B 0,C 180,E1 -26793.236,E2 -26793.236} C_VEL
LIN {X 0,Y 174.155,Z 363.151,A -85,B 0,C 180,E1 -26796.537,E2 -26796.537} C_VEL
LIN {X 0,Y 172.524,Z 358.706,A -85,B 0,C 180,E1 -26799.577,E2 -26799.577} C_VEL
LIN {X 0,Y 171.804,Z 357.172,A -85,B 0,C 180,E1 -26801.141,E2 -26801.141} C_VEL
LIN {X 0,Y 170.492,Z 354.047,A -85,B 0,C 180,E1 -26805.06,E2 -26805.06} C_VEL
LIN {X 0,Y 169.633,Z 352.746,A -85,B 0,C 180,E1 -26810.45,E2 -26810.45} C_VEL
LIN {X 0,Y 170.201,Z 353.349,A -85,B 0,C 180,E1 -26815.904,E2 -26815.904} C_VEL
LIN {X 0,Y 170.718,Z 353.996,A -85,B 0,C 180,E1 -26817.807,E2 -26817.807} C_VEL
LIN {X 0,Y 172.343,Z 357.84,A -85,B 0,C 180,E1 -26822.18,E2 -26822.18} C_VEL
LIN {X 0,Y 174.569,Z 362.786,A -85,B 0,C 180,E1 -26826.128,E2 -26826.128} C_VEL
LIN {X 0,Y 176.283,Z 367.015,A -85,B 0,C 180,E1 -26828.587,E2 -26828.587} C_VEL
LIN {X 0,Y 176.528,Z 367.801,A -85,B 0,C 180,E1 -26828.945,E2 -26828.945} C_VEL
LIN {X 0,Y 174.226,Z 380.786,A -85,B 0,C 180,E1 -26829.437,E2 -26829.437} C_VEL
LIN {X 0,Y 170.883,Z 392.921,A -85,B 0,C 180,E1 -26830.13,E2 -26830.13} C_VEL
LIN {X 0,Y 166.51,Z 404.657,A -85,B 0,C 180,E1 -26831.086,E2 -26831.086} C_VEL
LIN {X 0,Y 161.016,Z 416.16,A -85,B 0,C 180,E1 -26832.352,E2 -26832.352} C_VEL
LIN {X 0,Y 154.765,Z 426.72,A -85,B 0,C 180,E1 -26833.912,E2 -26833.912} C_VEL
LIN {X 0,Y 147.919,Z 436.248,A -85,B 0,C 180,E1 -26835.816,E2 -26835.816} C_VEL
LIN {X 0,Y 140.56,Z 444.921,A -85,B 0,C 180,E1 -26838.192,E2 -26838.192} C_VEL
LIN {X 0,Y 132.224,Z 453.233,A -85,B 0,C 180,E1 -26841.356,E2 -26841.356} C_VEL
LIN {X 0,Y 124.08,Z 459.952,A -85,B 0,C 180,E1 -26845.005,E2 -26845.005} C_VEL
LIN {X 0,Y 115.967,Z 465.583,A -85,B 0,C 180,E1 -26849.562,E2 -26849.562} C_VEL
LIN {X 0,Y 109.902,Z 469.07,A -85,B 0,C 180,E1 -26853.763,E2 -26853.763} C_VEL
LIN {X 0,Y 105.861,Z 471.072,A -85,B 0,C 180,E1 -26857.185,E2 -26857.185} C_VEL
LIN {X 0,Y 102.225,Z 472.561,A -85,B 0,C 180,E1 -26860.863,E2 -26860.863} C_VEL
LIN {X 0,Y 98.569,Z 473.722,A -85,B 0,C 180,E1 -26865.451,E2 -26865.451} C_VEL
LIN {X 0,Y 94.1,Z 474.325,A -85,B 0,C 180,E1 -26873.308,E2 -26873.308} C_VEL
LIN {X 0,Y 92.41,Z 474.007,A -85,B 0,C 180,E1 -26877.833,E2 -26877.833} C_VEL
LIN {X 0,Y 91.2,Z 473.274,A -85,B 0,C 180,E1 -26882.458,E2 -26882.458} C_VEL
LIN {X 0,Y 90.423,Z 471.555,A -85,B 0,C 180,E1 -26888.794,E2 -26888.794} C_VEL
LIN {X 0,Y 90.53,Z 468.336,A -85,B 0,C 180,E1 -26896.531,E2 -26896.531} C_VEL
LIN {X 0,Y 91.771,Z 463.582,A -85,B 0,C 180,E1 -26904.371,E2 -26904.371} C_VEL
LIN {X 0,Y 93.763,Z 458.016,A -85,B 0,C 180,E1 -26911.072,E2 -26911.072} C_VEL
LIN {X 0,Y 96.595,Z 451.176,A -85,B 0,C 180,E1 -26917.314,E2 -26917.314} C_VEL
LIN {X 0,Y 100.406,Z 442.522,A -85,B 0,C 180,E1 -26923.251,E2 -26923.251} C_VEL
LIN {X 0,Y 104.126,Z 433.905,A -85,B 0,C 180,E1 -26927.68,E2 -26927.68} C_VEL
LIN {X 0,Y 108.541,Z 423.058,A -85,B 0,C 180,E1 -26931.857,E2 -26931.857} C_VEL
LIN {X 0,Y 112.43,Z 412.249,A -85,B 0,C 180,E1 -26934.956,E2 -26934.956} C_VEL
LIN {X 0,Y 116.04,Z 400.128,A -85,B 0,C 180,E1 -26937.502,E2 -26937.502} C_VEL
LIN {X 0,Y 118.932,Z 387.54,A -85,B 0,C 180,E1 -26939.418,E2 -26939.418} C_VEL
LIN {X 0,Y 121.05,Z 375.334,A -85,B 0,C 180,E1 -26940.651,E2 -26940.651} C_VEL
LIN {X 0,Y 122.549,Z 360.416,A -85,B 0,C 180,E1 -26941.538,E2 -26941.538} C_VEL
LIN {X 0,Y 125.197,Z 325.956,A -85,B 0,C 180,E1 -26943.153,E2 -26943.153} C_VEL
LIN {X 0,Y 123.513,Z 321.673,A -85,B 0,C 180,E1 -26944.252,E2 -26944.252} C_VEL
LIN {X 0,Y 118.756,Z 311.682,A -85,B 0,C 180,E1 -26947.443,E2 -26947.443} C_VEL
LIN {X 0,Y 113.528,Z 302.442,A -85,B 0,C 180,E1 -26951.348,E2 -26951.348} C_VEL
LIN {X 0,Y 108.435,Z 294.71,A -85,B 0,C 180,E1 -26955.759,E2 -26955.759} C_VEL
LIN {X 0,Y 105.791,Z 290.999,A -85,B 0,C 180,E1 -26958.394,E2 -26958.394} C_VEL
LIN {X 0,Y 103.232,Z 287.666,A -85,B 0,C 180,E1 -26961.243,E2 -26961.243} C_VEL
LIN {X 0,Y 102.464,Z 286.413,A -85,B 0,C 180,E1 -26962.216,E2 -26962.216} C_VEL
LIN {X 0,Y 99.939,Z 284.039,A -85,B 0,C 180,E1 -26965.484,E2 -26965.484} C_VEL
LIN {X 0,Y 98.295,Z 281.143,A -85,B 0,C 180,E1 -26968.184,E2 -26968.184} C_VEL
LIN {X 0,Y 95.25,Z 278.985,A -85,B 0,C 180,E1 -26973.746,E2 -26973.746} C_VEL
LIN {X 0,Y 93.835,Z 275.948,A -85,B 0,C 180,E1 -26978.607,E2 -26978.607} C_VEL
LIN {X 0,Y 93.82,Z 275.306,A -85,B 0,C 180,E1 -26982.585,E2 -26982.585} C_VEL
LIN {X 0,Y 94.084,Z 275.209,A -85,B 0,C 180,E1 -26987.071,E2 -26987.071} C_VEL
LIN {X 0,Y 94.196,Z 275.251,A -85,B 0,C 180,E1 -26991.438,E2 -26991.438} C_VEL
LIN {X 0,Y 94.771,Z 275.145,A -85,B 0,C 180,E1 -27000.019,E2 -27000.019} C_VEL
LIN {X 0,Y 94.381,Z 275.72,A -85,B 0,C 180,E1 -27004.289,E2 -27004.289} C_VEL
LIN {X 0,Y 94.802,Z 277.314,A -85,B 0,C 180,E1 -27006.671,E2 -27006.671} C_VEL
LIN {X 0,Y 96.74,Z 279.908,A -85,B 0,C 180,E1 -27011.012,E2 -27011.012} C_VEL
LIN {X 0,Y 98.767,Z 281.393,A -85,B 0,C 180,E1 -27014.356,E2 -27014.356} C_VEL
LIN {X 0,Y 100.372,Z 284.394,A -85,B 0,C 180,E1 -27016.937,E2 -27016.937} C_VEL
LIN {X 0,Y 102.891,Z 286.806,A -85,B 0,C 180,E1 -27020.118,E2 -27020.118} C_VEL
LIN {X 0,Y 105.023,Z 290.177,A -85,B 0,C 180,E1 -27022.648,E2 -27022.648} C_VEL
LIN {X 0,Y 106.364,Z 291.673,A -85,B 0,C 180,E1 -27024.02,E2 -27024.02} C_VEL
LIN {X 0,Y 109.852,Z 296.815,A -85,B 0,C 180,E1 -27027.383,E2 -27027.383} C_VEL
LIN {X 0,Y 113.657,Z 302.711,A -85,B 0,C 180,E1 -27030.591,E2 -27030.591} C_VEL
LIN {X 0,Y 118.944,Z 312.184,A -85,B 0,C 180,E1 -27034.532,E2 -27034.532} C_VEL
LIN {X 0,Y 121.387,Z 317.394,A -85,B 0,C 180,E1 -27036.219,E2 -27036.219} C_VEL
LIN {X 0,Y 124.781,Z 328.301,A -85,B 0,C 180,E1 -27038.686,E2 -27038.686} C_VEL
LIN {X 0,Y 125.029,Z 330.681,A -85,B 0,C 180,E1 -27038.983,E2 -27038.983} C_VEL
LIN {X 0,Y 121.573,Z 373.739,A -85,B 0,C 180,E1 -27041.09,E2 -27041.09} C_VEL
LIN {X 0,Y 119.485,Z 386.803,A -85,B 0,C 180,E1 -27042.207,E2 -27042.207} C_VEL
LIN {X 0,Y 116.938,Z 398.865,A -85,B 0,C 180,E1 -27043.848,E2 -27043.848} C_VEL
LIN {X 0,Y 113.675,Z 410.181,A -85,B 0,C 180,E1 -27045.932,E2 -27045.932} C_VEL
LIN {X 0,Y 110.551,Z 419.247,A -85,B 0,C 180,E1 -27048.127,E2 -27048.127} C_VEL
LIN {X 0,Y 106.846,Z 429.203,A -85,B 0,C 180,E1 -27051.328,E2 -27051.328} C_VEL
LIN {X 0,Y 103.512,Z 437.175,A -85,B 0,C 180,E1 -27054.588,E2 -27054.588} C_VEL
LIN {X 0,Y 99.745,Z 445.982,A -85,B 0,C 180,E1 -27059.282,E2 -27059.282} C_VEL
LIN {X 0,Y 96.071,Z 454.288,A -85,B 0,C 180,E1 -27065.127,E2 -27065.127} C_VEL
LIN {X 0,Y 93.71,Z 459.929,A -85,B 0,C 180,E1 -27070.278,E2 -27070.278} C_VEL
LIN {X 0,Y 91.9,Z 465.426,A -85,B 0,C 180,E1 -27076.738,E2 -27076.738} C_VEL
LIN {X 0,Y 91.001,Z 469.696,A -85,B 0,C 180,E1 -27083.349,E2 -27083.349} C_VEL
LIN {X 0,Y 90.939,Z 472.87,A -85,B 0,C 180,E1 -27090.001,E2 -27090.001} C_VEL
LIN {X 0,Y 90.939,Z 474.422,A -85,B 0,C 180,E1 -27094.434,E2 -27094.434} C_VEL
LIN {X 0,Y 91.275,Z 475.567,A -85,B 0,C 180,E1 -27098.86,E2 -27098.86} C_VEL
LIN {X 0,Y 93.352,Z 476.616,A -85,B 0,C 180,E1 -27107.528,E2 -27107.528} C_VEL
LIN {X 0,Y 97.234,Z 476.171,A -85,B 0,C 180,E1 -27115.702,E2 -27115.702} C_VEL
LIN {X 0,Y 99.971,Z 475.367,A -85,B 0,C 180,E1 -27119.48,E2 -27119.48} C_VEL
LIN {X 0,Y 106.622,Z 472.547,A -85,B 0,C 180,E1 -27126.388,E2 -27126.388} C_VEL
LIN {X 0,Y 112.573,Z 469.345,A -85,B 0,C 180,E1 -27130.961,E2 -27130.961} C_VEL
LIN {X 0,Y 119.012,Z 465.128,A -85,B 0,C 180,E1 -27135.125,E2 -27135.125} C_VEL
LIN {X 0,Y 127.379,Z 458.764,A -85,B 0,C 180,E1 -27139.346,E2 -27139.346} C_VEL
LIN {X 0,Y 135.158,Z 451.825,A -85,B 0,C 180,E1 -27142.466,E2 -27142.466} C_VEL
LIN {X 0,Y 143.304,Z 443.173,A -85,B 0,C 180,E1 -27145.233,E2 -27145.233} C_VEL
LIN {X 0,Y 150.262,Z 434.362,A -85,B 0,C 180,E1 -27147.342,E2 -27147.342} C_VEL
LIN {X 0,Y 156.79,Z 424.679,A -85,B 0,C 180,E1 -27149.012,E2 -27149.012} C_VEL
LIN {X 0,Y 162.698,Z 414.081,A -85,B 0,C 180,E1 -27150.382,E2 -27150.382} C_VEL
LIN {X 0,Y 167.948,Z 402.244,A -85,B 0,C 180,E1 -27151.495,E2 -27151.495} C_VEL
LIN {X 0,Y 171.408,Z 392.321,A -85,B 0,C 180,E1 -27152.201,E2 -27152.201} C_VEL
LIN {X 0,Y 173.079,Z 385.726,A -85,B 0,C 180,E1 -27152.743,E2 -27152.743} C_VEL
LIN {X 0,Y 173.815,Z 380.641,A -85,B 0,C 180,E1 -27153.431,E2 -27153.431} C_VEL
LIN {X 0,Y 173.919,Z 376.135,A -85,B 0,C 180,E1 -27154.414,E2 -27154.414} C_VEL
LIN {X 0,Y 173.548,Z 373.431,A -85,B 0,C 180,E1 -27155.392,E2 -27155.392} C_VEL
LIN {X 0,Y 172.112,Z 368.229,A -85,B 0,C 180,E1 -27158.271,E2 -27158.271} C_VEL
LIN {X 0,Y 170.918,Z 364.478,A -85,B 0,C 180,E1 -27161.04,E2 -27161.04} C_VEL
LIN {X 0,Y 169.445,Z 360.977,A -85,B 0,C 180,E1 -27165.58,E2 -27165.58} C_VEL
LIN {X 0,Y 168.738,Z 359.827,A -85,B 0,C 180,E1 -27170.399,E2 -27170.399} C_VEL
LIN {X 0,Y 169.301,Z 360.38,A -85,B 0,C 180,E1 -27175.882,E2 -27175.882} C_VEL
LIN {X 0,Y 169.659,Z 360.884,A -85,B 0,C 180,E1 -27177.292,E2 -27177.292} C_VEL
LIN {X 0,Y 171.125,Z 364.67,A -85,B 0,C 180,E1 -27181.607,E2 -27181.607} C_VEL
LIN {X 0,Y 173.065,Z 369.509,A -85,B 0,C 180,E1 -27185.524,E2 -27185.524} C_VEL
LIN {X 0,Y 173.829,Z 371.736,A -85,B 0,C 180,E1 -27186.883,E2 -27186.883} C_VEL
LIN {X 0,Y 170.848,Z 385.432,A -85,B 0,C 180,E1 -27187.423,E2 -27187.423} C_VEL
LIN {X 0,Y 167.034,Z 397.465,A -85,B 0,C 180,E1 -27188.16,E2 -27188.16} C_VEL
LIN {X 0,Y 161.973,Z 409.401,A -85,B 0,C 180,E1 -27189.201,E2 -27189.201} C_VEL
LIN {X 0,Y 155.529,Z 421.333,A -85,B 0,C 180,E1 -27190.628,E2 -27190.628} C_VEL
LIN {X 0,Y 148.388,Z 431.925,A -85,B 0,C 180,E1 -27192.35,E2 -27192.35} C_VEL
LIN {X 0,Y 140.315,Z 441.817,A -85,B 0,C 180,E1 -27194.632,E2 -27194.632} C_VEL
LIN {X 0,Y 132.432,Z 449.898,A -85,B 0,C 180,E1 -27197.205,E2 -27197.205} C_VEL
LIN {X 0,Y 123.71,Z 457.347,A -85,B 0,C 180,E1 -27200.578,E2 -27200.578} C_VEL
LIN {X 0,Y 115.729,Z 463.065,A -85,B 0,C 180,E1 -27204.365,E2 -27204.365} C_VEL
LIN {X 0,Y 108.2,Z 467.547,A -85,B 0,C 180,E1 -27208.73,E2 -27208.73} C_VEL
LIN {X 0,Y 101.417,Z 470.842,A -85,B 0,C 180,E1 -27213.737,E2 -27213.737} C_VEL
LIN {X 0,Y 97.383,Z 472.448,A -85,B 0,C 180,E1 -27217.451,E2 -27217.451} C_VEL
LIN {X 0,Y 92.58,Z 473.855,A -85,B 0,C 180,E1 -27223.066,E2 -27223.066} C_VEL
LIN {X 0,Y 88.1,Z 474.446,A -85,B 0,C 180,E1 -27230.342,E2 -27230.342} C_VEL
LIN {X 0,Y 86.067,Z 474.202,A -85,B 0,C 180,E1 -27235.137,E2 -27235.137} C_VEL
LIN {X 0,Y 84.549,Z 473.528,A -85,B 0,C 180,E1 -27240.081,E2 -27240.081} C_VEL
LIN {X 0,Y 83.387,Z 471.626,A -85,B 0,C 180,E1 -27247.922,E2 -27247.922} C_VEL
LIN {X 0,Y 83.335,Z 468.831,A -85,B 0,C 180,E1 -27255.343,E2 -27255.343} C_VEL
LIN {X 0,Y 84.298,Z 464.754,A -85,B 0,C 180,E1 -27263.055,E2 -27263.055} C_VEL
LIN {X 0,Y 86.111,Z 459.807,A -85,B 0,C 180,E1 -27269.998,E2 -27269.998} C_VEL
LIN {X 0,Y 88.886,Z 453.41,A -85,B 0,C 180,E1 -27276.81,E2 -27276.81} C_VEL
LIN {X 0,Y 92.621,Z 445.386,A -85,B 0,C 180,E1 -27283.156,E2 -27283.156} C_VEL
LIN {X 0,Y 96.697,Z 436.541,A -85,B 0,C 180,E1 -27288.389,E2 -27288.389} C_VEL
LIN {X 0,Y 100.936,Z 427.16,A -85,B 0,C 180,E1 -27292.515,E2 -27292.515} C_VEL
LIN {X 0,Y 104.949,Z 417.273,A -85,B 0,C 180,E1 -27295.801,E2 -27295.801} C_VEL
LIN {X 0,Y 108.636,Z 406.555,A -85,B 0,C 180,E1 -27298.495,E2 -27298.495} C_VEL
LIN {X 0,Y 112.174,Z 393.682,A -85,B 0,C 180,E1 -27300.86,E2 -27300.86} C_VEL
LIN {X 0,Y 114.927,Z 380.663,A -85,B 0,C 180,E1 -27302.477,E2 -27302.477} C_VEL
LIN {X 0,Y 116.763,Z 367.444,A -85,B 0,C 180,E1 -27303.473,E2 -27303.473} C_VEL
LIN {X 0,Y 120.026,Z 327.898,A -85,B 0,C 180,E1 -27305.37,E2 -27305.37} C_VEL
LIN {X 0,Y 114.933,Z 316.597,A -85,B 0,C 180,E1 -27309.091,E2 -27309.091} C_VEL
LIN {X 0,Y 110.144,Z 307.778,A -85,B 0,C 180,E1 -27313.014,E2 -27313.014} C_VEL
LIN {X 0,Y 105.58,Z 300.535,A -85,B 0,C 180,E1 -27317.353,E2 -27317.353} C_VEL
LIN {X 0,Y 102.976,Z 296.774,A -85,B 0,C 180,E1 -27320.194,E2 -27320.194} C_VEL
LIN {X 0,Y 100.492,Z 293.087,A -85,B 0,C 180,E1 -27323.327,E2 -27323.327} C_VEL
LIN {X 0,Y 97.66,Z 289.935,A -85,B 0,C 180,E1 -27327.385,E2 -27327.385} C_VEL
LIN {X 0,Y 96.562,Z 287.842,A -85,B 0,C 180,E1 -27329.395,E2 -27329.395} C_VEL
LIN {X 0,Y 93.815,Z 285.671,A -85,B 0,C 180,E1 -27334.902,E2 -27334.902} C_VEL
LIN {X 0,Y 92.291,Z 282.555,A -85,B 0,C 180,E1 -27339.982,E2 -27339.982} C_VEL
LIN {X 0,Y 91.012,Z 281.63,A -85,B 0,C 180,E1 -27346.626,E2 -27346.626} C_VEL
LIN {X 0,Y 91.895,Z 281.634,A -85,B 0,C 180,E1 -27360.02,E2 -27360.02} C_VEL
LIN {X 0,Y 92.92,Z 282.775,A -85,B 0,C 180,E1 -27363.814,E2 -27363.814} C_VEL
LIN {X 0,Y 94.804,Z 286.229,A -85,B 0,C 180,E1 -27369.082,E2 -27369.082} C_VEL
LIN {X 0,Y 96.897,Z 288.06,A -85,B 0,C 180,E1 -27372.989,E2 -27372.989} C_VEL
LIN {X 0,Y 98.697,Z 291.174,A -85,B 0,C 180,E1 -27376.041,E2 -27376.041} C_VEL
LIN {X 0,Y 100.661,Z 293.288,A -85,B 0,C 180,E1 -27378.725,E2 -27378.725} C_VEL
LIN {X 0,Y 103.299,Z 297.094,A -85,B 0,C 180,E1 -27381.992,E2 -27381.992} C_VEL
LIN {X 0,Y 106.914,Z 302.628,A -85,B 0,C 180,E1 -27385.834,E2 -27385.834} C_VEL
LIN {X 0,Y 110.392,Z 308.33,A -85,B 0,C 180,E1 -27389.048,E2 -27389.048} C_VEL
LIN {X 0,Y 115.288,Z 317.509,A -85,B 0,C 180,E1 -27393.03,E2 -27393.03} C_VEL
LIN {X 0,Y 117.299,Z 322.277,A -85,B 0,C 180,E1 -27394.581,E2 -27394.581} C_VEL
LIN {X 0,Y 119.869,Z 331.083,A -85,B 0,C 180,E1 -27396.66,E2 -27396.66} C_VEL
LIN {X 0,Y 116.309,Z 373.75,A -85,B 0,C 180,E1 -27398.796,E2 -27398.796} C_VEL
LIN {X 0,Y 114.07,Z 387.216,A -85,B 0,C 180,E1 -27399.98,E2 -27399.98} C_VEL
LIN {X 0,Y 111.231,Z 399.665,A -85,B 0,C 180,E1 -27401.726,E2 -27401.726} C_VEL
LIN {X 0,Y 107.558,Z 411.552,A -85,B 0,C 180,E1 -27404.05,E2 -27404.05} C_VEL
LIN {X 0,Y 104.796,Z 419.027,A -85,B 0,C 180,E1 -27405.912,E2 -27405.912} C_VEL
LIN {X 0,Y 100.874,Z 429.016,A -85,B 0,C 180,E1 -27409.221,E2 -27409.221} C_VEL
LIN {X 0,Y 97.258,Z 437.133,A -85,B 0,C 180,E1 -27412.671,E2 -27412.671} C_VEL
LIN {X 0,Y 92.903,Z 446.574,A -85,B 0,C 180,E1 -27418.028,E2 -27418.028} C_VEL
LIN {X 0,Y 89.037,Z 454.761,A -85,B 0,C 180,E1 -27424.272,E2 -27424.272} C_VEL
LIN {X 0,Y 86.237,Z 461.321,A -85,B 0,C 180,E1 -27430.976,E2 -27430.976} C_VEL
LIN {X 0,Y 84.519,Z 466.499,A -85,B 0,C 180,E1 -27438.003,E2 -27438.003} C_VEL
LIN {X 0,Y 83.824,Z 470.489,A -85,B 0,C 180,E1 -27445.192,E2 -27445.192} C_VEL
LIN {X 0,Y 83.839,Z 472.526,A -85,B 0,C 180,E1 -27450.002,E2 -27450.002} C_VEL
LIN {X 0,Y 83.879,Z 474.122,A -85,B 0,C 180,E1 -27454.808,E2 -27454.808} C_VEL
LIN {X 0,Y 85.208,Z 476.113,A -85,B 0,C 180,E1 -27464.328,E2 -27464.328} C_VEL
LIN {X 0,Y 88.488,Z 476.502,A -85,B 0,C 180,E1 -27473.4,E2 -27473.4} C_VEL
LIN {X 0,Y 93.843,Z 475.408,A -85,B 0,C 180,E1 -27481.619,E2 -27481.619} C_VEL
LIN {X 0,Y 97.261,Z 474.259,A -85,B 0,C 180,E1 -27485.317,E2 -27485.317} C_VEL
LIN {X 0,Y 100.986,Z 472.703,A -85,B 0,C 180,E1 -27488.782,E2 -27488.782} C_VEL
LIN {X 0,Y 107.305,Z 469.601,A -85,B 0,C 180,E1 -27493.45,E2 -27493.45} C_VEL
LIN {X 0,Y 114.125,Z 465.488,A -85,B 0,C 180,E1 -27497.646,E2 -27497.646} C_VEL
LIN {X 0,Y 122.882,Z 459.238,A -85,B 0,C 180,E1 -27501.852,E2 -27501.852} C_VEL
LIN {X 0,Y 130.976,Z 452.444,A -85,B 0,C 180,E1 -27504.916,E2 -27504.916} C_VEL
LIN {X 0,Y 137.959,Z 445.536,A -85,B 0,C 180,E1 -27507.2,E2 -27507.2} C_VEL
LIN {X 0,Y 145.133,Z 437.251,A -85,B 0,C 180,E1 -27509.266,E2 -27509.266} C_VEL
LIN {X 0,Y 152.537,Z 427.063,A -85,B 0,C 180,E1 -27511.094,E2 -27511.094} C_VEL
LIN {X 0,Y 159.351,Z 415.602,A -85,B 0,C 180,E1 -27512.573,E2 -27512.573} C_VEL
LIN {X 0,Y 164.724,Z 404.33,A -85,B 0,C 180,E1 -27513.635,E2 -27513.635} C_VEL
LIN {X 0,Y 169.145,Z 392.19,A -85,B 0,C 180,E1 -27514.474,E2 -27514.474} C_VEL
LIN {X 0,Y 172.733,Z 378.34,A -85,B 0,C 180,E1 -27515.127,E2 -27515.127} C_VEL
LIN {X 0,Y 173.569,Z 373.521,A -85,B 0,C 180,E1 -27515.349,E2 -27515.349} C_VEL
LIN {X 0,Y 173.548,Z 373.431,A -85,B 0,C 180,E1 -27515.392,E2 -27515.392} C_VEL
LIN {X 0,Y 172.608,Z 370.824,A -85,B 0,C 180,E1 -27517.118,E2 -27517.118} C_VEL
LIN {X 0,Y 171.496,Z 369.398,A -85,B 0,C 180,E1 -27519.007,E2 -27519.007} C_VEL
LIN {X 0,Y 169.387,Z 368.51,A -85,B 0,C 180,E1 -27523.032,E2 -27523.032} C_VEL
LIN {X 0,Y 168.44,Z 367.998,A -85,B 0,C 180,E1 -27525.791,E2 -27525.791} C_VEL
LIN {X 0,Y 167.818,Z 366.904,A -85,B 0,C 180,E1 -27530.346,E2 -27530.346} C_VEL
LIN {X 0,Y 168.211,Z 367.312,A -85,B 0,C 180,E1 -27535.196,E2 -27535.196} C_VEL
LIN {X 0,Y 168.594,Z 367.914,A -85,B 0,C 180,E1 -27536.95,E2 -27536.95} C_VEL
LIN {X 0,Y 169.693,Z 371.228,A -85,B 0,C 180,E1 -27540.842,E2 -27540.842} C_VEL
LIN {X 0,Y 171.172,Z 375.897,A -85,B 0,C 180,E1 -27544.699,E2 -27544.699} C_VEL
LIN {X 0,Y 167.843,Z 389.111,A -85,B 0,C 180,E1 -27545.311,E2 -27545.311} C_VEL
LIN {X 0,Y 163.182,Z 402.03,A -85,B 0,C 180,E1 -27546.133,E2 -27546.133} C_VEL
LIN {X 0,Y 157.619,Z 413.729,A -85,B 0,C 180,E1 -27547.205,E2 -27547.205} C_VEL
LIN {X 0,Y 150.762,Z 425.14,A -85,B 0,C 180,E1 -27548.642,E2 -27548.642} C_VEL
LIN {X 0,Y 142.939,Z 435.703,A -85,B 0,C 180,E1 -27550.465,E2 -27550.465} C_VEL
LIN {X 0,Y 135.035,Z 444.494,A -85,B 0,C 180,E1 -27552.613,E2 -27552.613} C_VEL
LIN {X 0,Y 125.841,Z 453.021,A -85,B 0,C 180,E1 -27555.551,E2 -27555.551} C_VEL
LIN {X 0,Y 118.451,Z 458.735,A -85,B 0,C 180,E1 -27558.316,E2 -27558.316} C_VEL
LIN {X 0,Y 108.9,Z 464.918,A -85,B 0,C 180,E1 -27562.762,E2 -27562.762} C_VEL
LIN {X 0,Y 99.756,Z 469.603,A -85,B 0,C 180,E1 -27568.277,E2 -27568.277} C_VEL
LIN {X 0,Y 92.932,Z 472.287,A -85,B 0,C 180,E1 -27573.706,E2 -27573.706} C_VEL
LIN {X 0,Y 86.769,Z 473.989,A -85,B 0,C 180,E1 -27580.359,E2 -27580.359} C_VEL
LIN {X 0,Y 82.375,Z 474.523,A -85,B 0,C 180,E1 -27586.956,E2 -27586.956} C_VEL
LIN {X 0,Y 79.78,Z 474.357,A -85,B 0,C 180,E1 -27592.41,E2 -27592.41} C_VEL
LIN {X 0,Y 78.084,Z 473.781,A -85,B 0,C 180,E1 -27597.312,E2 -27597.312} C_VEL
LIN {X 0,Y 76.342,Z 471.681,A -85,B 0,C 180,E1 -27606.947,E2 -27606.947} C_VEL
LIN {X 0,Y 76.332,Z 468.198,A -85,B 0,C 180,E1 -27616.691,E2 -27616.691} C_VEL
LIN {X 0,Y 77.566,Z 463.878,A -85,B 0,C 180,E1 -27625.017,E2 -27625.017} C_VEL
LIN {X 0,Y 80.19,Z 457.595,A -85,B 0,C 180,E1 -27633.767,E2 -27633.767} C_VEL
LIN {X 0,Y 83.539,Z 450.626,A -85,B 0,C 180,E1 -27640.91,E2 -27640.91} C_VEL
LIN {X 0,Y 87.137,Z 443.505,A -85,B 0,C 180,E1 -27646.395,E2 -27646.395} C_VEL
LIN {X 0,Y 91.596,Z 434.571,A -85,B 0,C 180,E1 -27651.57,E2 -27651.57} C_VEL
LIN {X 0,Y 96.38,Z 424.216,A -85,B 0,C 180,E1 -27655.944,E2 -27655.944} C_VEL
LIN {X 0,Y 100.679,Z 413.623,A -85,B 0,C 180,E1 -27659.25,E2 -27659.25} C_VEL
LIN {X 0,Y 104.693,Z 401.935,A -85,B 0,C 180,E1 -27661.912,E2 -27661.912} C_VEL
LIN {X 0,Y 107.869,Z 389.844,A -85,B 0,C 180,E1 -27663.907,E2 -27663.907} C_VEL
LIN {X 0,Y 110.491,Z 376.566,A -85,B 0,C 180,E1 -27665.357,E2 -27665.357} C_VEL
LIN {X 0,Y 112.026,Z 364.14,A -85,B 0,C 180,E1 -27666.172,E2 -27666.172} C_VEL
LIN {X 0,Y 114.929,Z 330.26,A -85,B 0,C 180,E1 -27667.789,E2 -27667.789} C_VEL
LIN {X 0,Y 110.787,Z 320.755,A -85,B 0,C 180,E1 -27671.193,E2 -27671.193} C_VEL
LIN {X 0,Y 106.724,Z 312.885,A -85,B 0,C 180,E1 -27674.914,E2 -27674.914} C_VEL
LIN {X 0,Y 102.471,Z 305.793,A -85,B 0,C 180,E1 -27679.417,E2 -27679.417} C_VEL
LIN {X 0,Y 100.465,Z 302.799,A -85,B 0,C 180,E1 -27681.846,E2 -27681.846} C_VEL
LIN {X 0,Y 97.996,Z 299.073,A -85,B 0,C 180,E1 -27685.29,E2 -27685.29} C_VEL
LIN {X 0,Y 95.482,Z 295.84,A -85,B 0,C 180,E1 -27689.386,E2 -27689.386} C_VEL
LIN {X 0,Y 94.807,Z 294.516,A -85,B 0,C 180,E1 -27690.768,E2 -27690.768} C_VEL
LIN {X 0,Y 92.349,Z 292.247,A -85,B 0,C 180,E1 -27696.292,E2 -27696.292} C_VEL
LIN {X 0,Y 91.007,Z 289.302,A -85,B 0,C 180,E1 -27701.447,E2 -27701.447} C_VEL
LIN {X 0,Y 89.902,Z 288.521,A -85,B 0,C 180,E1 -27711.026,E2 -27711.026} C_VEL
LIN {X 0,Y 91.181,Z 288.929,A -85,B 0,C 180,E1 -27720.863,E2 -27720.863} C_VEL
LIN {X 0,Y 91.625,Z 289.575,A -85,B 0,C 180,E1 -27722.615,E2 -27722.615} C_VEL
LIN {X 0,Y 93.532,Z 293.137,A -85,B 0,C 180,E1 -27728.39,E2 -27728.39} C_VEL
LIN {X 0,Y 95.051,Z 294.567,A -85,B 0,C 180,E1 -27731.481,E2 -27731.481} C_VEL
LIN {X 0,Y 97.127,Z 298.029,A -85,B 0,C 180,E1 -27735.24,E2 -27735.24} C_VEL
LIN {X 0,Y 98.586,Z 299.8,A -85,B 0,C 180,E1 -27737.387,E2 -27737.387} C_VEL
LIN {X 0,Y 101.728,Z 304.691,A -85,B 0,C 180,E1 -27741.55,E2 -27741.55} C_VEL
LIN {X 0,Y 104.253,Z 308.74,A -85,B 0,C 180,E1 -27744.405,E2 -27744.405} C_VEL
LIN {X 0,Y 107.256,Z 313.999,A -85,B 0,C 180,E1 -27747.451,E2 -27747.451} C_VEL
LIN {X 0,Y 111.465,Z 322.314,A -85,B 0,C 180,E1 -27751.229,E2 -27751.229} C_VEL
LIN {X 0,Y 113.025,Z 326.357,A -85,B 0,C 180,E1 -27752.582,E2 -27752.582} C_VEL
LIN {X 0,Y 114.856,Z 332.943,A -85,B 0,C 180,E1 -27754.253,E2 -27754.253} C_VEL
LIN {X 0,Y 111.3,Z 373.266,A -85,B 0,C 180,E1 -27756.276,E2 -27756.276} C_VEL
LIN {X 0,Y 108.951,Z 386.777,A -85,B 0,C 180,E1 -27757.442,E2 -27757.442} C_VEL
LIN {X 0,Y 105.997,Z 399.284,A -85,B 0,C 180,E1 -27759.204,E2 -27759.204} C_VEL
LIN {X 0,Y 102.139,Z 411.239,A -85,B 0,C 180,E1 -27761.56,E2 -27761.56} C_VEL
LIN {X 0,Y 99.215,Z 418.73,A -85,B 0,C 180,E1 -27763.445,E2 -27763.445} C_VEL
LIN {X 0,Y 95.055,Z 428.769,A -85,B 0,C 180,E1 -27766.852,E2 -27766.852} C_VEL
LIN {X 0,Y 90.763,Z 437.799,A -85,B 0,C 180,E1 -27770.893,E2 -27770.893} C_VEL
LIN {X 0,Y 86.94,Z 445.625,A -85,B 0,C 180,E1 -27775.54,E2 -27775.54} C_VEL
LIN {X 0,Y 82.681,Z 453.958,A -85,B 0,C 180,E1 -27782.129,E2 -27782.129} C_VEL
LIN {X 0,Y 79.517,Z 460.646,A -85,B 0,C 180,E1 -27789.298,E2 -27789.298} C_VEL
LIN {X 0,Y 77.581,Z 465.956,A -85,B 0,C 180,E1 -27796.912,E2 -27796.912} C_VEL
LIN {X 0,Y 76.763,Z 470.052,A -85,B 0,C 180,E1 -27804.749,E2 -27804.749} C_VEL
LIN {X 0,Y 76.762,Z 472.173,A -85,B 0,C 180,E1 -27810.002,E2 -27810.002} C_VEL
LIN {X 0,Y 76.804,Z 473.816,A -85,B 0,C 180,E1 -27815.252,E2 -27815.252} C_VEL
LIN {X 0,Y 78.326,Z 475.916,A -85,B 0,C 180,E1 -27825.617,E2 -27825.617} C_VEL
LIN {X 0,Y 79.882,Z 476.372,A -85,B 0,C 180,E1 -27830.606,E2 -27830.606} C_VEL
LIN {X 0,Y 84.632,Z 476.111,A -85,B 0,C 180,E1 -27839.886,E2 -27839.886} C_VEL
LIN {X 0,Y 91.54,Z 474.358,A -85,B 0,C 180,E1 -27847.895,E2 -27847.895} C_VEL
LIN {X 0,Y 95.553,Z 472.86,A -85,B 0,C 180,E1 -27851.451,E2 -27851.451} C_VEL
LIN {X 0,Y 102.262,Z 469.857,A -85,B 0,C 180,E1 -27856.19,E2 -27856.19} C_VEL
LIN {X 0,Y 109.479,Z 465.847,A -85,B 0,C 180,E1 -27860.386,E2 -27860.386} C_VEL
LIN {X 0,Y 117.304,Z 460.708,A -85,B 0,C 180,E1 -27863.982,E2 -27863.982} C_VEL
LIN {X 0,Y 125.618,Z 454.266,A -85,B 0,C 180,E1 -27867.058,E2 -27867.058} C_VEL
LIN {X 0,Y 134.265,Z 446.279,A -85,B 0,C 180,E1 -27869.734,E2 -27869.734} C_VEL
LIN {X 0,Y 141.67,Z 438.157,A -85,B 0,C 180,E1 -27871.71,E2 -27871.71} C_VEL
LIN {X 0,Y 149.274,Z 428.263,A -85,B 0,C 180,E1 -27873.451,E2 -27873.451} C_VEL
LIN {X 0,Y 156.235,Z 417.108,A -85,B 0,C 180,E1 -27874.864,E2 -27874.864} C_VEL
LIN {X 0,Y 162.23,Z 405.111,A -85,B 0,C 180,E1 -27875.95,E2 -27875.95} C_VEL
LIN {X 0,Y 166.604,Z 393.828,A -85,B 0,C 180,E1 -27876.695,E2 -27876.695} C_VEL
LIN {X 0,Y 170.132,Z 381.384,A -85,B 0,C 180,E1 -27877.286,E2 -27877.286} C_VEL
LIN {X 0,Y 170.989,Z 377.419,A -85,B 0,C 180,E1 -27877.463,E2 -27877.463} C_VEL
LIN {X 0,Y 170.013,Z 372.773,A -85,B 0,C 180,E1 -27880.364,E2 -27880.364} C_VEL
LIN {X 0,Y 169.342,Z 370.664,A -85,B 0,C 180,E1 -27882.365,E2 -27882.365} C_VEL
LIN {X 0,Y 168.44,Z 367.998,A -85,B 0,C 180,E1 -27885.791,E2 -27885.791} C_VEL
LIN {X 0,Y 167.966,Z 367.974,A -85,B 0,C 180,E1 -27887.8,E2 -27887.8} C_VEL
LIN {X 0,Y 167.552,Z 368.94,A -85,B 0,C 180,E1 -27889.798,E2 -27889.798} C_VEL
LIN {X 0,Y 167.228,Z 374.695,A -85,B 0,C 180,E1 -27896.403,E2 -27896.403} C_VEL
LIN {X 0,Y 168.011,Z 378.101,A -85,B 0,C 180,E1 -27900.401,E2 -27900.401} C_VEL
LIN {X 0,Y 168.592,Z 380.463,A -85,B 0,C 180,E1 -27902.527,E2 -27902.527} C_VEL
LIN {X 0,Y 164.892,Z 393.207,A -85,B 0,C 180,E1 -27903.144,E2 -27903.144} C_VEL
LIN {X 0,Y 160.262,Z 404.779,A -85,B 0,C 180,E1 -27903.912,E2 -27903.912} C_VEL
LIN {X 0,Y 154.311,Z 416.356,A -85,B 0,C 180,E1 -27904.961,E2 -27904.961} C_VEL
LIN {X 0,Y 147.588,Z 426.859,A -85,B 0,C 180,E1 -27906.25,E2 -27906.25} C_VEL
LIN {X 0,Y 140.112,Z 436.395,A -85,B 0,C 180,E1 -27907.84,E2 -27907.84} C_VEL
LIN {X 0,Y 131.974,Z 445.067,A -85,B 0,C 180,E1 -27909.872,E2 -27909.872} C_VEL
LIN {X 0,Y 122.466,Z 453.51,A -85,B 0,C 180,E1 -27912.684,E2 -27912.684} C_VEL
LIN {X 0,Y 113.274,Z 460.148,A -85,B 0,C 180,E1 -27915.909,E2 -27915.909} C_VEL
LIN {X 0,Y 104.549,Z 465.355,A -85,B 0,C 180,E1 -27919.758,E2 -27919.758} C_VEL
LIN {X 0,Y 96.371,Z 469.308,A -85,B 0,C 180,E1 -27924.273,E2 -27924.273} C_VEL
LIN {X 0,Y 88.922,Z 472.12,A -85,B 0,C 180,E1 -27929.61,E2 -27929.61} C_VEL
LIN {X 0,Y 81.159,Z 474.126,A -85,B 0,C 180,E1 -27937.283,E2 -27937.283} C_VEL
LIN {X 0,Y 76.954,Z 474.598,A -85,B 0,C 180,E1 -27943.06,E2 -27943.06} C_VEL
LIN {X 0,Y 73.338,Z 474.437,A -85,B 0,C 180,E1 -27950.012,E2 -27950.012} C_VEL
LIN {X 0,Y 70.21,Z 473.06,A -85,B 0,C 180,E1 -27959.965,E2 -27959.965} C_VEL
LIN {X 0,Y 69.305,Z 471.661,A -85,B 0,C 180,E1 -27966.067,E2 -27966.067} C_VEL
LIN {X 0,Y 69.127,Z 468.694,A -85,B 0,C 180,E1 -27975.274,E2 -27975.274} C_VEL
LIN {X 0,Y 70.468,Z 464.015,A -85,B 0,C 180,E1 -27985.446,E2 -27985.446} C_VEL
LIN {X 0,Y 72.96,Z 458.411,A -85,B 0,C 180,E1 -27994.141,E2 -27994.141} C_VEL
LIN {X 0,Y 76.475,Z 451.596,A -85,B 0,C 180,E1 -28001.931,E2 -28001.931} C_VEL
LIN {X 0,Y 81.118,Z 443.131,A -85,B 0,C 180,E1 -28008.957,E2 -28008.957} C_VEL
LIN {X 0,Y 85.786,Z 434.386,A -85,B 0,C 180,E1 -28014.179,E2 -28014.179} C_VEL
LIN {X 0,Y 91.051,Z 423.584,A -85,B 0,C 180,E1 -28018.842,E2 -28018.842} C_VEL
LIN {X 0,Y 95.66,Z 412.826,A -85,B 0,C 180,E1 -28022.183,E2 -28022.183} C_VEL
LIN {X 0,Y 99.874,Z 400.81,A -85,B 0,C 180,E1 -28024.87,E2 -28024.87} C_VEL
LIN {X 0,Y 103.261,Z 388.329,A -85,B 0,C 180,E1 -28026.852,E2 -28026.852} C_VEL
LIN {X 0,Y 105.797,Z 375.736,A -85,B 0,C 180,E1 -28028.161,E2 -28028.161} C_VEL
LIN {X 0,Y 107.432,Z 361.912,A -85,B 0,C 180,E1 -28029.016,E2 -28029.016} C_VEL
LIN {X 0,Y 110.074,Z 332.56,A -85,B 0,C 180,E1 -28030.414,E2 -28030.414} C_VEL
LIN {X 0,Y 106.32,Z 323.872,A -85,B 0,C 180,E1 -28033.925,E2 -28033.925} C_VEL
LIN {X 0,Y 102.82,Z 316.884,A -85,B 0,C 180,E1 -28037.606,E2 -28037.606} C_VEL
LIN {X 0,Y 99.45,Z 311.026,A -85,B 0,C 180,E1 -28041.668,E2 -28041.668} C_VEL
LIN {X 0,Y 97.048,Z 307.27,A -85,B 0,C 180,E1 -28045.041,E2 -28045.041} C_VEL
LIN {X 0,Y 95.789,Z 305.275,A -85,B 0,C 180,E1 -28047.049,E2 -28047.049} C_VEL
LIN {X 0,Y 93.369,Z 301.573,A -85,B 0,C 180,E1 -28051.621,E2 -28051.621} C_VEL
LIN {X 0,Y 90.713,Z 298.363,A -85,B 0,C 180,E1 -28058.523,E2 -28058.523} C_VEL
LIN {X 0,Y 89.891,Z 296.209,A -85,B 0,C 180,E1 -28062.387,E2 -28062.387} C_VEL
LIN {X 0,Y 89.009,Z 295.57,A -85,B 0,C 180,E1 -28070.935,E2 -28070.935} C_VEL
LIN {X 0,Y 90.076,Z 295.83,A -85,B 0,C 180,E1 -28080.02,E2 -28080.02} C_VEL
LIN {X 0,Y 90.411,Z 296.465,A -85,B 0,C 180,E1 -28081.564,E2 -28081.564} C_VEL
LIN {X 0,Y 92.098,Z 299.833,A -85,B 0,C 180,E1 -28087.253,E2 -28087.253} C_VEL
LIN {X 0,Y 93.334,Z 301.175,A -85,B 0,C 180,E1 -28090.047,E2 -28090.047} C_VEL
LIN {X 0,Y 95.574,Z 304.86,A -85,B 0,C 180,E1 -28094.404,E2 -28094.404} C_VEL
LIN {X 0,Y 96.559,Z 306.303,A -85,B 0,C 180,E1 -28096.003,E2 -28096.003} C_VEL
LIN {X 0,Y 99.544,Z 311.164,A -85,B 0,C 180,E1 -28100.285,E2 -28100.285} C_VEL
LIN {X 0,Y 102.818,Z 316.924,A -85,B 0,C 180,E1 -28104.231,E2 -28104.231} C_VEL
LIN {X 0,Y 106.585,Z 324.461,A -85,B 0,C 180,E1 -28108.169,E2 -28108.169} C_VEL
LIN {X 0,Y 108.701,Z 329.612,A -85,B 0,C 180,E1 -28110.216,E2 -28110.216} C_VEL
LIN {X 0,Y 110.042,Z 334.827,A -85,B 0,C 180,E1 -28111.631,E2 -28111.631} C_VEL
LIN {X 0,Y 106.442,Z 373.285,A -85,B 0,C 180,E1 -28113.553,E2 -28113.553} C_VEL
LIN {X 0,Y 103.958,Z 386.964,A -85,B 0,C 180,E1 -28114.741,E2 -28114.741} C_VEL
LIN {X 0,Y 100.692,Z 399.94,A -85,B 0,C 180,E1 -28116.618,E2 -28116.618} C_VEL
LIN {X 0,Y 96.299,Z 412.513,A -85,B 0,C 180,E1 -28119.159,E2 -28119.159} C_VEL
LIN {X 0,Y 93.31,Z 419.831,A -85,B 0,C 180,E1 -28121.136,E2 -28121.136} C_VEL
LIN {X 0,Y 88.915,Z 429.62,A -85,B 0,C 180,E1 -28124.656,E2 -28124.656} C_VEL
LIN {X 0,Y 84.744,Z 437.733,A -85,B 0,C 180,E1 -28128.438,E2 -28128.438} C_VEL
LIN {X 0,Y 80.261,Z 446.174,A -85,B 0,C 180,E1 -28133.77,E2 -28133.77} C_VEL
LIN {X 0,Y 75.739,Z 454.396,A -85,B 0,C 180,E1 -28140.848,E2 -28140.848} C_VEL
LIN {X 0,Y 72.878,Z 459.968,A -85,B 0,C 180,E1 -28147.312,E2 -28147.312} C_VEL
LIN {X 0,Y 70.65,Z 465.394,A -85,B 0,C 180,E1 -28155.602,E2 -28155.602} C_VEL
LIN {X 0,Y 69.682,Z 469.599,A -85,B 0,C 180,E1 -28164.213,E2 -28164.213} C_VEL
LIN {X 0,Y 69.674,Z 471.81,A -85,B 0,C 180,E1 -28170.002,E2 -28170.002} C_VEL
LIN {X 0,Y 69.752,Z 473.511,A -85,B 0,C 180,E1 -28175.785,E2 -28175.785} C_VEL
LIN {X 0,Y 71.5,Z 475.703,A -85,B 0,C 180,E1 -28187.152,E2 -28187.152} C_VEL
LIN {X 0,Y 73.255,Z 476.229,A -85,B 0,C 180,E1 -28192.568,E2 -28192.568} C_VEL
LIN {X 0,Y 78.548,Z 476.08,A -85,B 0,C 180,E1 -28202.471,E2 -28202.471} C_VEL
LIN {X 0,Y 86.03,Z 474.424,A -85,B 0,C 180,E1 -28210.811,E2 -28210.811} C_VEL
LIN {X 0,Y 90.354,Z 473.013,A -85,B 0,C 180,E1 -28214.432,E2 -28214.432} C_VEL
LIN {X 0,Y 98.509,Z 469.594,A -85,B 0,C 180,E1 -28219.83,E2 -28219.83} C_VEL
LIN {X 0,Y 107.783,Z 464.609,A -85,B 0,C 180,E1 -28224.595,E2 -28224.595} C_VEL
LIN {X 0,Y 116.116,Z 459.185,A -85,B 0,C 180,E1 -28227.928,E2 -28227.928} C_VEL
LIN {X 0,Y 124.907,Z 452.418,A -85,B 0,C 180,E1 -28230.707,E2 -28230.707} C_VEL
LIN {X 0,Y 133.884,Z 444.039,A -85,B 0,C 180,E1 -28233.176,E2 -28233.176} C_VEL
LIN {X 0,Y 141.561,Z 435.464,A -85,B 0,C 180,E1 -28234.967,E2 -28234.967} C_VEL
LIN {X 0,Y 149.427,Z 424.918,A -85,B 0,C 180,E1 -28236.514,E2 -28236.514} C_VEL
LIN {X 0,Y 155.8,Z 414.465,A -85,B 0,C 180,E1 -28237.63,E2 -28237.63} C_VEL
LIN {X 0,Y 161.23,Z 403.334,A -85,B 0,C 180,E1 -28238.517,E2 -28238.517} C_VEL
LIN {X 0,Y 166.033,Z 390.346,A -85,B 0,C 180,E1 -28239.264,E2 -28239.264} C_VEL
LIN {X 0,Y 168.489,Z 381.427,A -85,B 0,C 180,E1 -28239.67,E2 -28239.67} C_VEL
LIN {X 0,Y 167.925,Z 377.852,A -85,B 0,C 180,E1 -28242.326,E2 -28242.326} C_VEL
LIN {X 0,Y 167.161,Z 374.954,A -85,B 0,C 180,E1 -28246,E2 -28246} C_VEL
LIN {X 0,Y 166.637,Z 373.924,A -85,B 0,C 180,E1 -28250.277,E2 -28250.277} C_VEL
LIN {X 0,Y 166.889,Z 374.203,A -85,B 0,C 180,E1 -28254.552,E2 -28254.552} C_VEL
LIN {X 0,Y 167.228,Z 374.695,A -85,B 0,C 180,E1 -28256.403,E2 -28256.403} C_VEL
LIN {X 0,Y 167.279,Z 376.42,A -85,B 0,C 180,E1 -28257.673,E2 -28257.673} C_VEL
LIN {X 0,Y 167.028,Z 379.183,A -85,B 0,C 180,E1 -28258.727,E2 -28258.727} C_VEL
LIN {X 0,Y 166.229,Z 383.841,A -85,B 0,C 180,E1 -28259.796,E2 -28259.796} C_VEL
LIN {X 0,Y 164.887,Z 389.091,A -85,B 0,C 180,E1 -28260.475,E2 -28260.475} C_VEL
LIN {X 0,Y 164.037,Z 391.807,A -85,B 0,C 180,E1 -28260.65,E2 -28260.65} C_VEL
LIN {X 0,Y 159.055,Z 404.307,A -85,B 0,C 180,E1 -28261.368,E2 -28261.368} C_VEL
LIN {X 0,Y 152.97,Z 416.015,A -85,B 0,C 180,E1 -28262.329,E2 -28262.329} C_VEL
LIN {X 0,Y 146.105,Z 426.585,A -85,B 0,C 180,E1 -28263.498,E2 -28263.498} C_VEL
LIN {X 0,Y 139.288,Z 435.231,A -85,B 0,C 180,E1 -28264.773,E2 -28264.773} C_VEL
LIN {X 0,Y 130.711,Z 444.311,A -85,B 0,C 180,E1 -28266.667,E2 -28266.667} C_VEL
LIN {X 0,Y 121.03,Z 452.742,A -85,B 0,C 180,E1 -28269.186,E2 -28269.186} C_VEL
LIN {X 0,Y 111.438,Z 459.586,A -85,B 0,C 180,E1 -28272.164,E2 -28272.164} C_VEL
LIN {X 0,Y 101.499,Z 465.296,A -85,B 0,C 180,E1 -28276.06,E2 -28276.06} C_VEL
LIN {X 0,Y 93.496,Z 469.014,A -85,B 0,C 180,E1 -28280.009,E2 -28280.009} C_VEL
LIN {X 0,Y 85.398,Z 471.953,A -85,B 0,C 180,E1 -28285.138,E2 -28285.138} C_VEL
LIN {X 0,Y 80.455,Z 473.31,A -85,B 0,C 180,E1 -28289.125,E2 -28289.125} C_VEL
LIN {X 0,Y 75.808,Z 474.26,A -85,B 0,C 180,E1 -28293.766,E2 -28293.766} C_VEL
LIN {X 0,Y 71.955,Z 474.674,A -85,B 0,C 180,E1 -28298.61,E2 -28298.61} C_VEL
LIN {X 0,Y 67.106,Z 474.522,A -85,B 0,C 180,E1 -28307.105,E2 -28307.105} C_VEL
LIN {X 0,Y 63.773,Z 473.373,A -85,B 0,C 180,E1 -28316.561,E2 -28316.561} C_VEL
LIN {X 0,Y 62.357,Z 471.798,A -85,B 0,C 180,E1 -28324.303,E2 -28324.303} C_VEL
LIN {X 0,Y 61.967,Z 469.185,A -85,B 0,C 180,E1 -28333.526,E2 -28333.526} C_VEL
LIN {X 0,Y 62.892,Z 465.264,A -85,B 0,C 180,E1 -28343.582,E2 -28343.582} C_VEL
LIN {X 0,Y 65.217,Z 460.175,A -85,B 0,C 180,E1 -28353.087,E2 -28353.087} C_VEL
LIN {X 0,Y 68.743,Z 453.792,A -85,B 0,C 180,E1 -28361.797,E2 -28361.797} C_VEL
LIN {X 0,Y 73.444,Z 445.799,A -85,B 0,C 180,E1 -28369.566,E2 -28369.566} C_VEL
LIN {X 0,Y 78.318,Z 437.331,A -85,B 0,C 180,E1 -28375.468,E2 -28375.468} C_VEL
LIN {X 0,Y 83.679,Z 427.619,A -85,B 0,C 180,E1 -28380.258,E2 -28380.258} C_VEL
LIN {X 0,Y 88.455,Z 417.771,A -85,B 0,C 180,E1 -28383.789,E2 -28383.789} C_VEL
LIN {X 0,Y 92.81,Z 407.123,A -85,B 0,C 180,E1 -28386.606,E2 -28386.606} C_VEL
LIN {X 0,Y 96.959,Z 394.325,A -85,B 0,C 180,E1 -28389.026,E2 -28389.026} C_VEL
LIN {X 0,Y 100.13,Z 381.485,A -85,B 0,C 180,E1 -28390.647,E2 -28390.647} C_VEL
LIN {X 0,Y 102.196,Z 368.961,A -85,B 0,C 180,E1 -28391.616,E2 -28391.616} C_VEL
LIN {X 0,Y 105.432,Z 335.035,A -85,B 0,C 180,E1 -28393.283,E2 -28393.283} C_VEL
LIN {X 0,Y 102.224,Z 327.201,A -85,B 0,C 180,E1 -28396.771,E2 -28396.771} C_VEL
LIN {X 0,Y 99.115,Z 320.855,A -85,B 0,C 180,E1 -28400.541,E2 -28400.541} C_VEL
LIN {X 0,Y 95.967,Z 315.124,A -85,B 0,C 180,E1 -28405.015,E2 -28405.015} C_VEL
LIN {X 0,Y 93.8,Z 311.584,A -85,B 0,C 180,E1 -28408.676,E2 -28408.676} C_VEL
LIN {X 0,Y 91.456,Z 307.794,A -85,B 0,C 180,E1 -28413.702,E2 -28413.702} C_VEL
LIN {X 0,Y 89.39,Z 304.931,A -85,B 0,C 180,E1 -28420.016,E2 -28420.016} C_VEL
LIN {X 0,Y 88.797,Z 303.139,A -85,B 0,C 180,E1 -28423.349,E2 -28423.349} C_VEL
LIN {X 0,Y 88.117,Z 302.619,A -85,B 0,C 180,E1 -28430.843,E2 -28430.843} C_VEL
LIN {X 0,Y 89.031,Z 302.835,A -85,B 0,C 180,E1 -28439.401,E2 -28439.401} C_VEL
LIN {X 0,Y 91.045,Z 306.936,A -85,B 0,C 180,E1 -28447.003,E2 -28447.003} C_VEL
LIN {X 0,Y 91.782,Z 307.97,A -85,B 0,C 180,E1 -28448.829,E2 -28448.829} C_VEL
LIN {X 0,Y 94.521,Z 312.64,A -85,B 0,C 180,E1 -28454.429,E2 -28454.429} C_VEL
LIN {X 0,Y 96.992,Z 316.929,A -85,B 0,C 180,E1 -28458.364,E2 -28458.364} C_VEL
LIN {X 0,Y 100.043,Z 322.693,A -85,B 0,C 180,E1 -28462.475,E2 -28462.475} C_VEL
LIN {X 0,Y 103.663,Z 330.644,A -85,B 0,C 180,E1 -28466.682,E2 -28466.682} C_VEL
LIN {X 0,Y 105.011,Z 334.616,A -85,B 0,C 180,E1 -28468.19,E2 -28468.19} C_VEL
LIN {X 0,Y 105.427,Z 336.336,A -85,B 0,C 180,E1 -28468.695,E2 -28468.695} C_VEL
LIN {X 0,Y 101.833,Z 373.461,A -85,B 0,C 180,E1 -28470.596,E2 -28470.596} C_VEL
LIN {X 0,Y 99.381,Z 386.405,A -85,B 0,C 180,E1 -28471.693,E2 -28471.693} C_VEL
LIN {X 0,Y 96.249,Z 398.493,A -85,B 0,C 180,E1 -28473.371,E2 -28473.371} C_VEL
LIN {X 0,Y 91.963,Z 410.607,A -85,B 0,C 180,E1 -28475.713,E2 -28475.713} C_VEL
LIN {X 0,Y 88.142,Z 419.553,A -85,B 0,C 180,E1 -28478.062,E2 -28478.062} C_VEL
LIN {X 0,Y 83.407,Z 429.484,A -85,B 0,C 180,E1 -28481.692,E2 -28481.692} C_VEL
LIN {X 0,Y 78.793,Z 437.835,A -85,B 0,C 180,E1 -28485.705,E2 -28485.705} C_VEL
LIN {X 0,Y 73.68,Z 446.725,A -85,B 0,C 180,E1 -28491.686,E2 -28491.686} C_VEL
LIN {X 0,Y 68.849,Z 454.835,A -85,B 0,C 180,E1 -28499.312,E2 -28499.312} C_VEL
LIN {X 0,Y 65.324,Z 461.308,A -85,B 0,C 180,E1 -28507.882,E2 -28507.882} C_VEL
LIN {X 0,Y 63.224,Z 466.416,A -85,B 0,C 180,E1 -28517.157,E2 -28517.157} C_VEL
LIN {X 0,Y 62.53,Z 470.349,A -85,B 0,C 180,E1 -28526.781,E2 -28526.781} C_VEL
LIN {X 0,Y 62.577,Z 471.411,A -85,B 0,C 180,E1 -28530.002,E2 -28530.002} C_VEL
LIN {X 0,Y 62.685,Z 473.203,A -85,B 0,C 180,E1 -28536.439,E2 -28536.439} C_VEL
LIN {X 0,Y 64.745,Z 475.49,A -85,B 0,C 180,E1 -28549.007,E2 -28549.007} C_VEL
LIN {X 0,Y 69.37,Z 476.26,A -85,B 0,C 180,E1 -28560.437,E2 -28560.437} C_VEL
LIN {X 0,Y 76.507,Z 475.455,A -85,B 0,C 180,E1 -28570.02,E2 -28570.02} C_VEL
LIN {X 0,Y 85.431,Z 473.134,A -85,B 0,C 180,E1 -28577.766,E2 -28577.766} C_VEL
LIN {X 0,Y 93.545,Z 470.07,A -85,B 0,C 180,E1 -28582.849,E2 -28582.849} C_VEL
LIN {X 0,Y 101.022,Z 466.482,A -85,B 0,C 180,E1 -28586.6,E2 -28586.6} C_VEL
LIN {X 0,Y 109.573,Z 461.584,A -85,B 0,C 180,E1 -28589.986,E2 -28589.986} C_VEL
LIN {X 0,Y 118.544,Z 455.441,A -85,B 0,C 180,E1 -28592.786,E2 -28592.786} C_VEL
LIN {X 0,Y 127.734,Z 447.826,A -85,B 0,C 180,E1 -28595.211,E2 -28595.211} C_VEL
LIN {X 0,Y 137.132,Z 438.311,A -85,B 0,C 180,E1 -28597.296,E2 -28597.296} C_VEL
LIN {X 0,Y 145.153,Z 428.5,A -85,B 0,C 180,E1 -28598.758,E2 -28598.758} C_VEL
LIN {X 0,Y 152.445,Z 417.499,A -85,B 0,C 180,E1 -28599.94,E2 -28599.94} C_VEL
LIN {X 0,Y 158.957,Z 405.09,A -85,B 0,C 180,E1 -28600.886,E2 -28600.886} C_VEL
LIN {X 0,Y 163.778,Z 393.094,A -85,B 0,C 180,E1 -28601.549,E2 -28601.549} C_VEL
LIN {X 0,Y 166.037,Z 385.695,A -85,B 0,C 180,E1 -28601.915,E2 -28601.915} C_VEL
LIN {X 0,Y 165.815,Z 383.989,A -85,B 0,C 180,E1 -28603.523,E2 -28603.523} C_VEL
LIN {X 0,Y 165.46,Z 381.76,A -85,B 0,C 180,E1 -28606.479,E2 -28606.479} C_VEL
LIN {X 0,Y 165.079,Z 380.885,A -85,B 0,C 180,E1 -28610.184,E2 -28610.184} C_VEL
LIN {X 0,Y 165.228,Z 381,A -85,B 0,C 180,E1 -28613.885,E2 -28613.885} C_VEL
LIN {X 0,Y 165.534,Z 381.546,A -85,B 0,C 180,E1 -28616.033,E2 -28616.033} C_VEL
LIN {X 0,Y 165.955,Z 384.662,A -85,B 0,C 180,E1 -28619.762,E2 -28619.762} C_VEL
LIN {X 0,Y 166.04,Z 385.278,A -85,B 0,C 180,E1 -28620.335,E2 -28620.335} C_VEL
LIN {X 0,Y 164.037,Z 391.807,A -85,B 0,C 180,E1 -28620.65,E2 -28620.65} C_VEL
LIN {X 0,Y 161.968,Z 397.354,A -85,B 0,C 180,E1 -28620.693,E2 -28620.693} C_VEL
LIN {X 0,Y 157.661,Z 406.206,A -85,B 0,C 180,E1 -28620.21,E2 -28620.21} C_VEL
LIN {X 0,Y 152.677,Z 414.68,A -85,B 0,C 180,E1 -28619.809,E2 -28619.809} C_VEL
LIN {X 0,Y 149.529,Z 419.627,A -85,B 0,C 180,E1 -28620.016,E2 -28620.016} C_VEL
LIN {X 0,Y 141.474,Z 430.864,A -85,B 0,C 180,E1 -28621.26,E2 -28621.26} C_VEL
LIN {X 0,Y 133.676,Z 439.745,A -85,B 0,C 180,E1 -28622.642,E2 -28622.642} C_VEL
LIN {X 0,Y 125.12,Z 447.84,A -85,B 0,C 180,E1 -28624.415,E2 -28624.415} C_VEL
LIN {X 0,Y 114.564,Z 456.026,A -85,B 0,C 180,E1 -28627.031,E2 -28627.031} C_VEL
LIN {X 0,Y 103.615,Z 462.819,A -85,B 0,C 180,E1 -28630.414,E2 -28630.414} C_VEL
LIN {X 0,Y 94.206,Z 467.44,A -85,B 0,C 180,E1 -28634.106,E2 -28634.106} C_VEL
LIN {X 0,Y 83.591,Z 471.429,A -85,B 0,C 180,E1 -28639.628,E2 -28639.628} C_VEL
LIN {X 0,Y 77.018,Z 473.208,A -85,B 0,C 180,E1 -28644.141,E2 -28644.141} C_VEL
LIN {X 0,Y 70.796,Z 474.389,A -85,B 0,C 180,E1 -28649.728,E2 -28649.728} C_VEL
LIN {X 0,Y 63.464,Z 474.811,A -85,B 0,C 180,E1 -28659.176,E2 -28659.176} C_VEL
LIN {X 0,Y 60.175,Z 474.452,A -85,B 0,C 180,E1 -28665.509,E2 -28665.509} C_VEL
LIN {X 0,Y 57.578,Z 473.675,A -85,B 0,C 180,E1 -28672.386,E2 -28672.386} C_VEL
LIN {X 0,Y 55.446,Z 471.862,A -85,B 0,C 180,E1 -28682.457,E2 -28682.457} C_VEL
LIN {X 0,Y 54.922,Z 468.554,A -85,B 0,C 180,E1 -28695.169,E2 -28695.169} C_VEL
LIN {X 0,Y 56.287,Z 464.289,A -85,B 0,C 180,E1 -28706.623,E2 -28706.623} C_VEL
LIN {X 0,Y 59.682,Z 457.971,A -85,B 0,C 180,E1 -28718.462,E2 -28718.462} C_VEL
LIN {X 0,Y 64.023,Z 451.02,A -85,B 0,C 180,E1 -28727.568,E2 -28727.568} C_VEL
LIN {X 0,Y 69.588,Z 442.453,A -85,B 0,C 180,E1 -28735.291,E2 -28735.291} C_VEL
LIN {X 0,Y 75.188,Z 433.356,A -85,B 0,C 180,E1 -28740.935,E2 -28740.935} C_VEL
LIN {X 0,Y 80.646,Z 423.497,A -85,B 0,C 180,E1 -28745.262,E2 -28745.262} C_VEL
LIN {X 0,Y 85.809,Z 412.681,A -85,B 0,C 180,E1 -28748.644,E2 -28748.644} C_VEL
LIN {X 0,Y 90.496,Z 400.554,A -85,B 0,C 180,E1 -28751.307,E2 -28751.307} C_VEL
LIN {X 0,Y 94.19,Z 388.271,A -85,B 0,C 180,E1 -28753.174,E2 -28753.174} C_VEL
LIN {X 0,Y 96.961,Z 375.534,A -85,B 0,C 180,E1 -28754.44,E2 -28754.44} C_VEL
LIN {X 0,Y 98.873,Z 360.411,A -85,B 0,C 180,E1 -28755.299,E2 -28755.299} C_VEL
LIN {X 0,Y 101.092,Z 337.556,A -85,B 0,C 180,E1 -28756.39,E2 -28756.39} C_VEL
LIN {X 0,Y 97.909,Z 329.565,A -85,B 0,C 180,E1 -28760.477,E2 -28760.477} C_VEL
LIN {X 0,Y 94.507,Z 322.603,A -85,B 0,C 180,E1 -28765.543,E2 -28765.543} C_VEL
LIN {X 0,Y 91.916,Z 317.889,A -85,B 0,C 180,E1 -28770.33,E2 -28770.33} C_VEL
LIN {X 0,Y 89.837,Z 314.371,A -85,B 0,C 180,E1 -28775.343,E2 -28775.343} C_VEL
LIN {X 0,Y 88.054,Z 311.223,A -85,B 0,C 180,E1 -28782.02,E2 -28782.02} C_VEL
LIN {X 0,Y 87.807,Z 310.174,A -85,B 0,C 180,E1 -28783.831,E2 -28783.831} C_VEL
LIN {X 0,Y 87.228,Z 309.643,A -85,B 0,C 180,E1 -28790.748,E2 -28790.748} C_VEL
LIN {X 0,Y 88.041,Z 309.986,A -85,B 0,C 180,E1 -28799.057,E2 -28799.057} C_VEL
LIN {X 0,Y 89.589,Z 313.597,A -85,B 0,C 180,E1 -28805.647,E2 -28805.647} C_VEL
LIN {X 0,Y 90.273,Z 314.718,A -85,B 0,C 180,E1 -28807.569,E2 -28807.569} C_VEL
LIN {X 0,Y 92.506,Z 318.825,A -85,B 0,C 180,E1 -28812.672,E2 -28812.672} C_VEL
LIN {X 0,Y 94.937,Z 323.422,A -85,B 0,C 180,E1 -28816.986,E2 -28816.986} C_VEL
LIN {X 0,Y 97.705,Z 329.245,A -85,B 0,C 180,E1 -28821.098,E2 -28821.098} C_VEL
LIN {X 0,Y 100.868,Z 337.087,A -85,B 0,C 180,E1 -28825.189,E2 -28825.189} C_VEL
LIN {X 0,Y 101.178,Z 338.41,A -85,B 0,C 180,E1 -28825.626,E2 -28825.626} C_VEL
LIN {X 0,Y 97.497,Z 373.808,A -85,B 0,C 180,E1 -28827.382,E2 -28827.382} C_VEL
LIN {X 0,Y 94.915,Z 386.686,A -85,B 0,C 180,E1 -28828.447,E2 -28828.447} C_VEL
LIN {X 0,Y 91.462,Z 399.192,A -85,B 0,C 180,E1 -28830.182,E2 -28830.182} C_VEL
LIN {X 0,Y 86.612,Z 411.884,A -85,B 0,C 180,E1 -28832.666,E2 -28832.666} C_VEL
LIN {X 0,Y 83.259,Z 419.274,A -85,B 0,C 180,E1 -28834.616,E2 -28834.616} C_VEL
LIN {X 0,Y 78.264,Z 429.128,A -85,B 0,C 180,E1 -28838.214,E2 -28838.214} C_VEL
LIN {X 0,Y 73.19,Z 437.73,A -85,B 0,C 180,E1 -28842.417,E2 -28842.417} C_VEL
LIN {X 0,Y 68.226,Z 445.774,A -85,B 0,C 180,E1 -28847.969,E2 -28847.969} C_VEL
LIN {X 0,Y 62.835,Z 454.032,A -85,B 0,C 180,E1 -28855.999,E2 -28855.999} C_VEL
LIN {X 0,Y 58.776,Z 460.653,A -85,B 0,C 180,E1 -28865.263,E2 -28865.263} C_VEL
LIN {X 0,Y 56.311,Z 465.897,A -85,B 0,C 180,E1 -28875.548,E2 -28875.548} C_VEL
LIN {X 0,Y 55.453,Z 469.934,A -85,B 0,C 180,E1 -28886.369,E2 -28886.369} C_VEL
LIN {X 0,Y 55.497,Z 471.01,A -85,B 0,C 180,E1 -28890.002,E2 -28890.002} C_VEL
LIN {X 0,Y 55.631,Z 472.865,A -85,B 0,C 180,E1 -28897.26,E2 -28897.26} C_VEL
LIN {X 0,Y 56.457,Z 474.28,A -85,B 0,C 180,E1 -28904.419,E2 -28904.419} C_VEL
LIN {X 0,Y 60.361,Z 475.894,A -85,B 0,C 180,E1 -28917.76,E2 -28917.76} C_VEL
LIN {X 0,Y 66.999,Z 476.012,A -85,B 0,C 180,E1 -28929.007,E2 -28929.007} C_VEL
LIN {X 0,Y 75.824,Z 474.549,A -85,B 0,C 180,E1 -28937.862,E2 -28937.862} C_VEL
LIN {X 0,Y 86.127,Z 471.556,A -85,B 0,C 180,E1 -28944.689,E2 -28944.689} C_VEL
LIN {X 0,Y 94.433,Z 468.182,A -85,B 0,C 180,E1 -28948.858,E2 -28948.858} C_VEL
LIN {X 0,Y 103.2,Z 463.773,A -85,B 0,C 180,E1 -28952.292,E2 -28952.292} C_VEL
LIN {X 0,Y 113.922,Z 457.129,A -85,B 0,C 180,E1 -28955.5,E2 -28955.5} C_VEL
LIN {X 0,Y 123.363,Z 449.914,A -85,B 0,C 180,E1 -28957.786,E2 -28957.786} C_VEL
LIN {X 0,Y 132.974,Z 440.997,A -85,B 0,C 180,E1 -28959.742,E2 -28959.742} C_VEL
LIN {X 0,Y 141.111,Z 431.813,A -85,B 0,C 180,E1 -28961.138,E2 -28961.138} C_VEL
LIN {X 0,Y 148.531,Z 421.616,A -85,B 0,C 180,E1 -28962.225,E2 -28962.225} C_VEL
LIN {X 0,Y 155.599,Z 409.551,A -85,B 0,C 180,E1 -28963.144,E2 -28963.144} C_VEL
LIN {X 0,Y 160.999,Z 397.604,A -85,B 0,C 180,E1 -28963.815,E2 -28963.815} C_VEL
LIN {X 0,Y 162.976,Z 392.216,A -85,B 0,C 180,E1 -28964.058,E2 -28964.058} C_VEL
LIN {X 0,Y 163.499,Z 390.315,A -85,B 0,C 180,E1 -28964.405,E2 -28964.405} C_VEL
LIN {X 0,Y 163.297,Z 388.313,A -85,B 0,C 180,E1 -28967.563,E2 -28967.563} C_VEL
LIN {X 0,Y 163.152,Z 387.653,A -85,B 0,C 180,E1 -28972.207,E2 -28972.207} C_VEL
LIN {X 0,Y 163.415,Z 387.992,A -85,B 0,C 180,E1 -28975.055,E2 -28975.055} C_VEL
LIN {X 0,Y 163.515,Z 390.03,A -85,B 0,C 180,E1 -28977.939,E2 -28977.939} C_VEL
LIN {X 0,Y 163.164,Z 391.293,A -85,B 0,C 180,E1 -28978.168,E2 -28978.168} C_VEL
LIN {X 0,Y 158.184,Z 403.801,A -85,B 0,C 180,E1 -28978.79,E2 -28978.79} C_VEL
LIN {X 0,Y 151.688,Z 416.131,A -85,B 0,C 180,E1 -28979.696,E2 -28979.696} C_VEL
LIN {X 0,Y 149.529,Z 419.627,A -85,B 0,C 180,E1 -28980.016,E2 -28980.016} C_VEL
LIN {X 0,Y 146.144,Z 424.528,A -85,B 0,C 180,E1 -28980.256,E2 -28980.256} C_VEL
LIN {X 0,Y 139.805,Z 432.196,A -85,B 0,C 180,E1 -28979.98,E2 -28979.98} C_VEL
LIN {X 0,Y 133.006,Z 439.288,A -85,B 0,C 180,E1 -28979.787,E2 -28979.787} C_VEL
LIN {X 0,Y 128.858,Z 443.274,A -85,B 0,C 180,E1 -28980.218,E2 -28980.218} C_VEL
LIN {X 0,Y 119.551,Z 451.232,A -85,B 0,C 180,E1 -28982.009,E2 -28982.009} C_VEL
LIN {X 0,Y 109.209,Z 458.424,A -85,B 0,C 180,E1 -28984.404,E2 -28984.404} C_VEL
LIN {X 0,Y 99.19,Z 464.054,A -85,B 0,C 180,E1 -28987.266,E2 -28987.266} C_VEL
LIN {X 0,Y 89.436,Z 468.413,A -85,B 0,C 180,E1 -28990.8,E2 -28990.8} C_VEL
LIN {X 0,Y 80.044,Z 471.62,A -85,B 0,C 180,E1 -28995.248,E2 -28995.248} C_VEL
LIN {X 0,Y 74.219,Z 473.116,A -85,B 0,C 180,E1 -28998.746,E2 -28998.746} C_VEL
LIN {X 0,Y 66.215,Z 474.516,A -85,B 0,C 180,E1 -29005.091,E2 -29005.091} C_VEL
LIN {X 0,Y 58.927,Z 474.946,A -85,B 0,C 180,E1 -29013.395,E2 -29013.395} C_VEL
LIN {X 0,Y 54.984,Z 474.646,A -85,B 0,C 180,E1 -29019.92,E2 -29019.92} C_VEL
LIN {X 0,Y 51.769,Z 473.929,A -85,B 0,C 180,E1 -29027.248,E2 -29027.248} C_VEL
LIN {X 0,Y 48.594,Z 471.92,A -85,B 0,C 180,E1 -29040.119,E2 -29040.119} C_VEL
LIN {X 0,Y 47.749,Z 469.049,A -85,B 0,C 180,E1 -29052.877,E2 -29052.877} C_VEL
LIN {X 0,Y 49.21,Z 464.427,A -85,B 0,C 180,E1 -29067.462,E2 -29067.462} C_VEL
LIN {X 0,Y 52.524,Z 458.788,A -85,B 0,C 180,E1 -29079.626,E2 -29079.626} C_VEL
LIN {X 0,Y 57.2,Z 451.989,A -85,B 0,C 180,E1 -29089.746,E2 -29089.746} C_VEL
LIN {X 0,Y 63.099,Z 443.755,A -85,B 0,C 180,E1 -29097.997,E2 -29097.997} C_VEL
LIN {X 0,Y 69.102,Z 434.833,A -85,B 0,C 180,E1 -29104.01,E2 -29104.01} C_VEL
LIN {X 0,Y 74.867,Z 425.255,A -85,B 0,C 180,E1 -29108.453,E2 -29108.453} C_VEL
LIN {X 0,Y 80.338,Z 414.786,A -85,B 0,C 180,E1 -29111.836,E2 -29111.836} C_VEL
LIN {X 0,Y 85.273,Z 403.331,A -85,B 0,C 180,E1 -29114.469,E2 -29114.469} C_VEL
LIN {X 0,Y 89.255,Z 391.394,A -85,B 0,C 180,E1 -29116.414,E2 -29116.414} C_VEL
LIN {X 0,Y 92.5,Z 378.192,A -85,B 0,C 180,E1 -29117.782,E2 -29117.782} C_VEL
LIN {X 0,Y 94.555,Z 364.913,A -85,B 0,C 180,E1 -29118.605,E2 -29118.605} C_VEL
LIN {X 0,Y 97.059,Z 340.161,A -85,B 0,C 180,E1 -29119.768,E2 -29119.768} C_VEL
LIN {X 0,Y 94.359,Z 333.219,A -85,B 0,C 180,E1 -29123.854,E2 -29123.854} C_VEL
LIN {X 0,Y 91.762,Z 327.439,A -85,B 0,C 180,E1 -29128.483,E2 -29128.483} C_VEL
LIN {X 0,Y 89.857,Z 323.831,A -85,B 0,C 180,E1 -29132.618,E2 -29132.618} C_VEL
LIN {X 0,Y 88.44,Z 321.071,A -85,B 0,C 180,E1 -29136.612,E2 -29136.612} C_VEL
LIN {X 0,Y 86.9,Z 317.896,A -85,B 0,C 180,E1 -29143.421,E2 -29143.421} C_VEL
LIN {X 0,Y 86.76,Z 317.128,A -85,B 0,C 180,E1 -29144.758,E2 -29144.758} C_VEL
LIN {X 0,Y 86.583,Z 316.673,A -85,B 0,C 180,E1 -29155.365,E2 -29155.365} C_VEL
LIN {X 0,Y 86.989,Z 317.125,A -85,B 0,C 180,E1 -29158.376,E2 -29158.376} C_VEL
LIN {X 0,Y 88.382,Z 320.491,A -85,B 0,C 180,E1 -29164.867,E2 -29164.867} C_VEL
LIN {X 0,Y 90.659,Z 325.205,A -85,B 0,C 180,E1 -29171.039,E2 -29171.039} C_VEL
LIN {X 0,Y 93.057,Z 330.205,A -85,B 0,C 180,E1 -29175.768,E2 -29175.768} C_VEL
LIN {X 0,Y 95.571,Z 336.321,A -85,B 0,C 180,E1 -29179.903,E2 -29179.903} C_VEL
LIN {X 0,Y 97.146,Z 340.593,A -85,B 0,C 180,E1 -29182.217,E2 -29182.217} C_VEL
LIN {X 0,Y 93.626,Z 373.293,A -85,B 0,C 180,E1 -29183.814,E2 -29183.814} C_VEL
LIN {X 0,Y 90.969,Z 386.167,A -85,B 0,C 180,E1 -29184.805,E2 -29184.805} C_VEL
LIN {X 0,Y 87.348,Z 398.808,A -85,B 0,C 180,E1 -29186.481,E2 -29186.481} C_VEL
LIN {X 0,Y 82.98,Z 409.978,A -85,B 0,C 180,E1 -29188.517,E2 -29188.517} C_VEL
LIN {X 0,Y 78.707,Z 418.988,A -85,B 0,C 180,E1 -29190.75,E2 -29190.75} C_VEL
LIN {X 0,Y 72.76,Z 429.974,A -85,B 0,C 180,E1 -29194.816,E2 -29194.816} C_VEL
LIN {X 0,Y 66.21,Z 440.122,A -85,B 0,C 180,E1 -29200.143,E2 -29200.143} C_VEL
LIN {X 0,Y 60.924,Z 447.83,A -85,B 0,C 180,E1 -29206.204,E2 -29206.204} C_VEL
LIN {X 0,Y 56.146,Z 454.47,A -85,B 0,C 180,E1 -29213.52,E2 -29213.52} C_VEL
LIN {X 0,Y 52.385,Z 459.976,A -85,B 0,C 180,E1 -29221.997,E2 -29221.997} C_VEL
LIN {X 0,Y 49.466,Z 465.34,A -85,B 0,C 180,E1 -29233.495,E2 -29233.495} C_VEL
LIN {X 0,Y 48.376,Z 469.484,A -85,B 0,C 180,E1 -29245.837,E2 -29245.837} C_VEL
LIN {X 0,Y 48.4,Z 470.608,A -85,B 0,C 180,E1 -29250.003,E2 -29250.003} C_VEL
LIN {X 0,Y 48.602,Z 472.512,A -85,B 0,C 180,E1 -29258.317,E2 -29258.317} C_VEL
LIN {X 0,Y 49.598,Z 474.003,A -85,B 0,C 180,E1 -29266.466,E2 -29266.466} C_VEL
LIN {X 0,Y 54.173,Z 475.726,A -85,B 0,C 180,E1 -29281.263,E2 -29281.263} C_VEL
LIN {X 0,Y 57.535,Z 476.018,A -85,B 0,C 180,E1 -29287.647,E2 -29287.647} C_VEL
LIN {X 0,Y 66.263,Z 475.49,A -85,B 0,C 180,E1 -29297.942,E2 -29297.942} C_VEL
LIN {X 0,Y 76.618,Z 473.371,A -85,B 0,C 180,E1 -29305.647,E2 -29305.647} C_VEL
LIN {X 0,Y 88.003,Z 469.686,A -85,B 0,C 180,E1 -29311.461,E2 -29311.461} C_VEL
LIN {X 0,Y 97.028,Z 465.743,A -85,B 0,C 180,E1 -29314.881,E2 -29314.881} C_VEL
LIN {X 0,Y 106.392,Z 460.695,A -85,B 0,C 180,E1 -29317.642,E2 -29317.642} C_VEL
LIN {X 0,Y 116.02,Z 454.362,A -85,B 0,C 180,E1 -29319.874,E2 -29319.874} C_VEL
LIN {X 0,Y 125.778,Z 446.495,A -85,B 0,C 180,E1 -29321.788,E2 -29321.788} C_VEL
LIN {X 0,Y 133.997,Z 438.515,A -85,B 0,C 180,E1 -29323.178,E2 -29323.178} C_VEL
LIN {X 0,Y 142.349,Z 428.777,A -85,B 0,C 180,E1 -29324.314,E2 -29324.314} C_VEL
LIN {X 0,Y 149.907,Z 417.927,A -85,B 0,C 180,E1 -29325.231,E2 -29325.231} C_VEL
LIN {X 0,Y 156.635,Z 405.648,A -85,B 0,C 180,E1 -29325.968,E2 -29325.968} C_VEL
LIN {X 0,Y 160.455,Z 396.893,A -85,B 0,C 180,E1 -29326.37,E2 -29326.37} C_VEL
LIN {X 0,Y 160.861,Z 395.59,A -85,B 0,C 180,E1 -29326.793,E2 -29326.793} C_VEL
LIN {X 0,Y 160.783,Z 394.502,A -85,B 0,C 180,E1 -29329.919,E2 -29329.919} C_VEL
LIN {X 0,Y 160.827,Z 394.337,A -85,B 0,C 180,E1 -29332.456,E2 -29332.456} C_VEL
LIN {X 0,Y 160.975,Z 394.811,A -85,B 0,C 180,E1 -29334.98,E2 -29334.98} C_VEL
LIN {X 0,Y 160.948,Z 395.22,A -85,B 0,C 180,E1 -29335.615,E2 -29335.615} C_VEL
LIN {X 0,Y 160.742,Z 395.883,A -85,B 0,C 180,E1 -29335.843,E2 -29335.843} C_VEL
LIN {X 0,Y 155.712,Z 407.267,A -85,B 0,C 180,E1 -29336.425,E2 -29336.425} C_VEL
LIN {X 0,Y 149.526,Z 418.235,A -85,B 0,C 180,E1 -29337.176,E2 -29337.176} C_VEL
LIN {X 0,Y 141.507,Z 429.498,A -85,B 0,C 180,E1 -29338.239,E2 -29338.239} C_VEL
LIN {X 0,Y 132.456,Z 439.769,A -85,B 0,C 180,E1 -29339.59,E2 -29339.59} C_VEL
LIN {X 0,Y 128.858,Z 443.274,A -85,B 0,C 180,E1 -29340.218,E2 -29340.218} C_VEL
LIN {X 0,Y 124.528,Z 447.135,A -85,B 0,C 180,E1 -29340.726,E2 -29340.726} C_VEL
LIN {X 0,Y 116.562,Z 453.057,A -85,B 0,C 180,E1 -29340.806,E2 -29340.806} C_VEL
LIN {X 0,Y 108.16,Z 458.345,A -85,B 0,C 180,E1 -29340.959,E2 -29340.959} C_VEL
LIN {X 0,Y 103.164,Z 461.159,A -85,B 0,C 180,E1 -29341.702,E2 -29341.702} C_VEL
LIN {X 0,Y 91.694,Z 466.741,A -85,B 0,C 180,E1 -29344.852,E2 -29344.852} C_VEL
LIN {X 0,Y 81.706,Z 470.435,A -85,B 0,C 180,E1 -29348.428,E2 -29348.428} C_VEL
LIN {X 0,Y 72.134,Z 473.007,A -85,B 0,C 180,E1 -29353.01,E2 -29353.01} C_VEL
LIN {X 0,Y 62.092,Z 474.645,A -85,B 0,C 180,E1 -29359.818,E2 -29359.818} C_VEL
LIN {X 0,Y 55.093,Z 475.051,A -85,B 0,C 180,E1 -29366.748,E2 -29366.748} C_VEL
LIN {X 0,Y 49.781,Z 474.755,A -85,B 0,C 180,E1 -29374.337,E2 -29374.337} C_VEL
LIN {X 0,Y 43.425,Z 473.096,A -85,B 0,C 180,E1 -29389.653,E2 -29389.653} C_VEL
LIN {X 0,Y 40.938,Z 470.603,A -85,B 0,C 180,E1 -29404.581,E2 -29404.581} C_VEL
LIN {X 0,Y 40.998,Z 467.058,A -85,B 0,C 180,E1 -29420.126,E2 -29420.126} C_VEL
LIN {X 0,Y 43.43,Z 462.384,A -85,B 0,C 180,E1 -29434.638,E2 -29434.638} C_VEL
LIN {X 0,Y 47.728,Z 456.451,A -85,B 0,C 180,E1 -29447.125,E2 -29447.125} C_VEL
LIN {X 0,Y 53.59,Z 449.032,A -85,B 0,C 180,E1 -29457.32,E2 -29457.32} C_VEL
LIN {X 0,Y 60.628,Z 439.83,A -85,B 0,C 180,E1 -29465.42,E2 -29465.42} C_VEL
LIN {X 0,Y 67.259,Z 430.248,A -85,B 0,C 180,E1 -29470.771,E2 -29470.771} C_VEL
LIN {X 0,Y 73.698,Z 419.552,A -85,B 0,C 180,E1 -29474.69,E2 -29474.69} C_VEL
LIN {X 0,Y 79.561,Z 407.649,A -85,B 0,C 180,E1 -29477.712,E2 -29477.712} C_VEL
LIN {X 0,Y 84.317,Z 395.219,A -85,B 0,C 180,E1 -29479.846,E2 -29479.846} C_VEL
LIN {X 0,Y 88.108,Z 381.871,A -85,B 0,C 180,E1 -29481.37,E2 -29481.37} C_VEL
LIN {X 0,Y 90.559,Z 368.716,A -85,B 0,C 180,E1 -29482.226,E2 -29482.226} C_VEL
LIN {X 0,Y 93.354,Z 343.056,A -85,B 0,C 180,E1 -29483.382,E2 -29483.382} C_VEL
LIN {X 0,Y 91.314,Z 337.431,A -85,B 0,C 180,E1 -29487.098,E2 -29487.098} C_VEL
LIN {X 0,Y 89.365,Z 332.743,A -85,B 0,C 180,E1 -29491.284,E2 -29491.284} C_VEL
LIN {X 0,Y 88.021,Z 329.902,A -85,B 0,C 180,E1 -29494.799,E2 -29494.799} C_VEL
LIN {X 0,Y 87.081,Z 327.762,A -85,B 0,C 180,E1 -29497.946,E2 -29497.946} C_VEL
LIN {X 0,Y 85.781,Z 324.457,A -85,B 0,C 180,E1 -29505.061,E2 -29505.061} C_VEL
LIN {X 0,Y 85.731,Z 324.052,A -85,B 0,C 180,E1 -29505.786,E2 -29505.786} C_VEL
LIN {X 0,Y 85.683,Z 323.716,A -85,B 0,C 180,E1 -29515.317,E2 -29515.317} C_VEL
LIN {X 0,Y 85.922,Z 324.054,A -85,B 0,C 180,E1 -29517.356,E2 -29517.356} C_VEL
LIN {X 0,Y 87.324,Z 327.93,A -85,B 0,C 180,E1 -29524.637,E2 -29524.637} C_VEL
LIN {X 0,Y 88.952,Z 331.744,A -85,B 0,C 180,E1 -29529.513,E2 -29529.513} C_VEL
LIN {X 0,Y 90.827,Z 336.165,A -85,B 0,C 180,E1 -29533.748,E2 -29533.748} C_VEL
LIN {X 0,Y 93.019,Z 342.141,A -85,B 0,C 180,E1 -29537.882,E2 -29537.882} C_VEL
LIN {X 0,Y 93.438,Z 343.354,A -85,B 0,C 180,E1 -29538.6,E2 -29538.6} C_VEL
LIN {X 0,Y 89.988,Z 373.696,A -85,B 0,C 180,E1 -29540.014,E2 -29540.014} C_VEL
LIN {X 0,Y 87.148,Z 386.721,A -85,B 0,C 180,E1 -29540.958,E2 -29540.958} C_VEL
LIN {X 0,Y 83.256,Z 399.449,A -85,B 0,C 180,E1 -29542.594,E2 -29542.594} C_VEL
LIN {X 0,Y 78.304,Z 411.243,A -85,B 0,C 180,E1 -29544.671,E2 -29544.671} C_VEL
LIN {X 0,Y 74.559,Z 418.688,A -85,B 0,C 180,E1 -29546.435,E2 -29546.435} C_VEL
LIN {X 0,Y 68.223,Z 429.72,A -85,B 0,C 180,E1 -29550.377,E2 -29550.377} C_VEL
LIN {X 0,Y 62.109,Z 438.547,A -85,B 0,C 180,E1 -29554.747,E2 -29554.747} C_VEL
LIN {X 0,Y 57.178,Z 445.368,A -85,B 0,C 180,E1 -29559.81,E2 -29559.81} C_VEL
LIN {X 0,Y 50.6,Z 453.662,A -85,B 0,C 180,E1 -29568.724,E2 -29568.724} C_VEL
LIN {X 0,Y 46.2,Z 459.293,A -85,B 0,C 180,E1 -29577.834,E2 -29577.834} C_VEL
LIN {X 0,Y 42.676,Z 464.773,A -85,B 0,C 180,E1 -29590.773,E2 -29590.773} C_VEL
LIN {X 0,Y 41.298,Z 469.024,A -85,B 0,C 180,E1 -29605.122,E2 -29605.122} C_VEL
LIN {X 0,Y 41.318,Z 470.2,A -85,B 0,C 180,E1 -29610.003,E2 -29610.003} C_VEL
LIN {X 0,Y 41.607,Z 472.15,A -85,B 0,C 180,E1 -29619.728,E2 -29619.728} C_VEL
LIN {X 0,Y 45.095,Z 474.831,A -85,B 0,C 180,E1 -29637.878,E2 -29637.878} C_VEL
LIN {X 0,Y 52.077,Z 475.894,A -85,B 0,C 180,E1 -29652.439,E2 -29652.439} C_VEL
LIN {X 0,Y 61.723,Z 475.474,A -85,B 0,C 180,E1 -29662.852,E2 -29662.852} C_VEL
LIN {X 0,Y 67.114,Z 474.695,A -85,B 0,C 180,E1 -29666.905,E2 -29666.905} C_VEL
LIN {X 0,Y 78.762,Z 471.907,A -85,B 0,C 180,E1 -29673.168,E2 -29673.168} C_VEL
LIN {X 0,Y 87.942,Z 468.745,A -85,B 0,C 180,E1 -29676.789,E2 -29676.789} C_VEL
LIN {X 0,Y 97.426,Z 464.562,A -85,B 0,C 180,E1 -29679.684,E2 -29679.684} C_VEL
LIN {X 0,Y 108.826,Z 458.231,A -85,B 0,C 180,E1 -29682.284,E2 -29682.284} C_VEL
LIN {X 0,Y 118.753,Z 451.354,A -85,B 0,C 180,E1 -29684.095,E2 -29684.095} C_VEL
LIN {X 0,Y 128.781,Z 442.775,A -85,B 0,C 180,E1 -29685.624,E2 -29685.624} C_VEL
LIN {X 0,Y 137.219,Z 434.01,A -85,B 0,C 180,E1 -29686.691,E2 -29686.691} C_VEL
LIN {X 0,Y 145.713,Z 423.244,A -85,B 0,C 180,E1 -29687.609,E2 -29687.609} C_VEL
LIN {X 0,Y 152.965,Z 411.638,A -85,B 0,C 180,E1 -29688.278,E2 -29688.278} C_VEL
LIN {X 0,Y 157.672,Z 402.284,A -85,B 0,C 180,E1 -29688.703,E2 -29688.703} C_VEL
LIN {X 0,Y 158.053,Z 401.147,A -85,B 0,C 180,E1 -29689.743,E2 -29689.743} C_VEL
LIN {X 0,Y 158.122,Z 401.017,A -85,B 0,C 180,E1 -29693.097,E2 -29693.097} C_VEL
LIN {X 0,Y 157.359,Z 402.86,A -85,B 0,C 180,E1 -29693.587,E2 -29693.587} C_VEL
LIN {X 0,Y 150.991,Z 414.904,A -85,B 0,C 180,E1 -29694.226,E2 -29694.226} C_VEL
LIN {X 0,Y 143.742,Z 425.743,A -85,B 0,C 180,E1 -29695.009,E2 -29695.009} C_VEL
LIN {X 0,Y 135.624,Z 435.604,A -85,B 0,C 180,E1 -29695.981,E2 -29695.981} C_VEL
LIN {X 0,Y 126.653,Z 444.484,A -85,B 0,C 180,E1 -29697.235,E2 -29697.235} C_VEL
LIN {X 0,Y 115.981,Z 453.069,A -85,B 0,C 180,E1 -29699.021,E2 -29699.021} C_VEL
LIN {X 0,Y 105.444,Z 459.906,A -85,B 0,C 180,E1 -29701.169,E2 -29701.169} C_VEL
LIN {X 0,Y 103.164,Z 461.159,A -85,B 0,C 180,E1 -29701.702,E2 -29701.702} C_VEL
LIN {X 0,Y 98.064,Z 463.772,A -85,B 0,C 180,E1 -29702.566,E2 -29702.566} C_VEL
LIN {X 0,Y 85.221,Z 468.936,A -85,B 0,C 180,E1 -29703.384,E2 -29703.384} C_VEL
LIN {X 0,Y 77.787,Z 471.187,A -85,B 0,C 180,E1 -29704.399,E2 -29704.399} C_VEL
LIN {X 0,Y 74.247,Z 472.067,A -85,B 0,C 180,E1 -29705.505,E2 -29705.505} C_VEL
LIN {X 0,Y 64.284,Z 474.084,A -85,B 0,C 180,E1 -29710.273,E2 -29710.273} C_VEL
LIN {X 0,Y 58.015,Z 474.817,A -85,B 0,C 180,E1 -29714.266,E2 -29714.266} C_VEL
LIN {X 0,Y 52.098,Z 475.129,A -85,B 0,C 180,E1 -29719.206,E2 -29719.206} C_VEL
LIN {X 0,Y 44.82,Z 474.83,A -85,B 0,C 180,E1 -29728.014,E2 -29728.014} C_VEL
LIN {X 0,Y 37.96,Z 473.398,A -85,B 0,C 180,E1 -29742.215,E2 -29742.215} C_VEL
LIN {X 0,Y 35.186,Z 471.948,A -85,B 0,C 180,E1 -29753.182,E2 -29753.182} C_VEL
LIN {X 0,Y 33.573,Z 468.872,A -85,B 0,C 180,E1 -29771.695,E2 -29771.695} C_VEL
LIN {X 0,Y 35.108,Z 464.587,A -85,B 0,C 180,E1 -29790.405,E2 -29790.405} C_VEL
LIN {X 0,Y 39.972,Z 458.292,A -85,B 0,C 180,E1 -29807.916,E2 -29807.916} C_VEL
LIN {X 0,Y 46.13,Z 451.342,A -85,B 0,C 180,E1 -29819.676,E2 -29819.676} C_VEL
LIN {X 0,Y 52.57,Z 443.94,A -85,B 0,C 180,E1 -29827.462,E2 -29827.462} C_VEL
LIN {X 0,Y 59.134,Z 435.679,A -85,B 0,C 180,E1 -29833.105,E2 -29833.105} C_VEL
LIN {X 0,Y 66.472,Z 425.05,A -85,B 0,C 180,E1 -29837.737,E2 -29837.737} C_VEL
LIN {X 0,Y 72.582,Z 414.503,A -85,B 0,C 180,E1 -29840.768,E2 -29840.768} C_VEL
LIN {X 0,Y 78.026,Z 402.93,A -85,B 0,C 180,E1 -29843.069,E2 -29843.069} C_VEL
LIN {X 0,Y 82.355,Z 390.952,A -85,B 0,C 180,E1 -29844.687,E2 -29844.687} C_VEL
LIN {X 0,Y 85.85,Z 377.588,A -85,B 0,C 180,E1 -29845.838,E2 -29845.838} C_VEL
LIN {X 0,Y 87.97,Z 364.455,A -85,B 0,C 180,E1 -29846.5,E2 -29846.5} C_VEL
LIN {X 0,Y 90.016,Z 346.053,A -85,B 0,C 180,E1 -29847.248,E2 -29847.248} C_VEL
LIN {X 0,Y 87.955,Z 339.92,A -85,B 0,C 180,E1 -29852.124,E2 -29852.124} C_VEL
LIN {X 0,Y 86.525,Z 336.432,A -85,B 0,C 180,E1 -29856.353,E2 -29856.353} C_VEL
LIN {X 0,Y 85.723,Z 334.359,A -85,B 0,C 180,E1 -29859.524,E2 -29859.524} C_VEL
LIN {X 0,Y 84.705,Z 330.965,A -85,B 0,C 180,E1 -29867.099,E2 -29867.099} C_VEL
LIN {X 0,Y 84.888,Z 330.934,A -85,B 0,C 180,E1 -29876.299,E2 -29876.299} C_VEL
LIN {X 0,Y 85.947,Z 334.6,A -85,B 0,C 180,E1 -29883.146,E2 -29883.146} C_VEL
LIN {X 0,Y 87.14,Z 337.797,A -85,B 0,C 180,E1 -29887.406,E2 -29887.406} C_VEL
LIN {X 0,Y 88.815,Z 342.43,A -85,B 0,C 180,E1 -29891.89,E2 -29891.89} C_VEL
LIN {X 0,Y 90.063,Z 346.342,A -85,B 0,C 180,E1 -29894.706,E2 -29894.706} C_VEL
LIN {X 0,Y 86.797,Z 373.647,A -85,B 0,C 180,E1 -29895.91,E2 -29895.91} C_VEL
LIN {X 0,Y 83.895,Z 386.475,A -85,B 0,C 180,E1 -29896.716,E2 -29896.716} C_VEL
LIN {X 0,Y 79.978,Z 398.906,A -85,B 0,C 180,E1 -29898.177,E2 -29898.177} C_VEL
LIN {X 0,Y 74.82,Z 410.802,A -85,B 0,C 180,E1 -29900.068,E2 -29900.068} C_VEL
LIN {X 0,Y 70.886,Z 418.279,A -85,B 0,C 180,E1 -29901.65,E2 -29901.65} C_VEL
LIN {X 0,Y 64.148,Z 429.381,A -85,B 0,C 180,E1 -29905.334,E2 -29905.334} C_VEL
LIN {X 0,Y 58.348,Z 437.355,A -85,B 0,C 180,E1 -29908.997,E2 -29908.997} C_VEL
LIN {X 0,Y 51.56,Z 445.856,A -85,B 0,C 180,E1 -29915.135,E2 -29915.135} C_VEL
LIN {X 0,Y 44.343,Z 454.048,A -85,B 0,C 180,E1 -29924.508,E2 -29924.508} C_VEL
LIN {X 0,Y 38.646,Z 460.61,A -85,B 0,C 180,E1 -29936.941,E2 -29936.941} C_VEL
LIN {X 0,Y 35.129,Z 465.789,A -85,B 0,C 180,E1 -29952.541,E2 -29952.541} C_VEL
LIN {X 0,Y 34.228,Z 469.773,A -85,B 0,C 180,E1 -29970.004,E2 -29970.004} C_VEL
LIN {X 0,Y 34.632,Z 471.778,A -85,B 0,C 180,E1 -29981.712,E2 -29981.712} C_VEL
LIN {X 0,Y 38.959,Z 474.564,A -85,B 0,C 180,E1 -30002.768,E2 -30002.768} C_VEL
LIN {X 0,Y 42.631,Z 475.374,A -85,B 0,C 180,E1 -30011.26,E2 -30011.26} C_VEL
LIN {X 0,Y 47.068,Z 475.771,A -85,B 0,C 180,E1 -30018.3,E2 -30018.3} C_VEL
LIN {X 0,Y 57.699,Z 475.449,A -85,B 0,C 180,E1 -30028.502,E2 -30028.502} C_VEL
LIN {X 0,Y 63.514,Z 474.734,A -85,B 0,C 180,E1 -30032.283,E2 -30032.283} C_VEL
LIN {X 0,Y 69.606,Z 473.619,A -85,B 0,C 180,E1 -30035.331,E2 -30035.331} C_VEL
LIN {X 0,Y 82.165,Z 470.148,A -85,B 0,C 180,E1 -30040.205,E2 -30040.205} C_VEL
LIN {X 0,Y 91.908,Z 466.419,A -85,B 0,C 180,E1 -30042.914,E2 -30042.914} C_VEL
LIN {X 0,Y 101.852,Z 461.606,A -85,B 0,C 180,E1 -30045.026,E2 -30045.026} C_VEL
LIN {X 0,Y 111.953,Z 455.555,A -85,B 0,C 180,E1 -30046.668,E2 -30046.668} C_VEL
LIN {X 0,Y 122.111,Z 448.07,A -85,B 0,C 180,E1 -30048.079,E2 -30048.079} C_VEL
LIN {X 0,Y 130.618,Z 440.455,A -85,B 0,C 180,E1 -30049.103,E2 -30049.103} C_VEL
LIN {X 0,Y 140.071,Z 430.11,A -85,B 0,C 180,E1 -30049.96,E2 -30049.96} C_VEL
LIN {X 0,Y 147.824,Z 419.618,A -85,B 0,C 180,E1 -30050.586,E2 -30050.586} C_VEL
LIN {X 0,Y 151.719,Z 413.391,A -85,B 0,C 180,E1 -30050.881,E2 -30050.881} C_VEL
LIN {X 0,Y 152.622,Z 411.753,A -85,B 0,C 180,E1 -30051.379,E2 -30051.379} C_VEL
LIN {X 0,Y 145.819,Z 422.542,A -85,B 0,C 180,E1 -30051.962,E2 -30051.962} C_VEL
LIN {X 0,Y 138.18,Z 432.315,A -85,B 0,C 180,E1 -30052.66,E2 -30052.66} C_VEL
LIN {X 0,Y 129.229,Z 441.656,A -85,B 0,C 180,E1 -30053.591,E2 -30053.591} C_VEL
LIN {X 0,Y 119.972,Z 449.604,A -85,B 0,C 180,E1 -30054.796,E2 -30054.796} C_VEL
LIN {X 0,Y 109.921,Z 456.683,A -85,B 0,C 180,E1 -30056.318,E2 -30056.318} C_VEL
LIN {X 0,Y 98.429,Z 463.135,A -85,B 0,C 180,E1 -30058.472,E2 -30058.472} C_VEL
LIN {X 0,Y 87.866,Z 467.751,A -85,B 0,C 180,E1 -30061.01,E2 -30061.01} C_VEL
LIN {X 0,Y 77.525,Z 471.18,A -85,B 0,C 180,E1 -30064.264,E2 -30064.264} C_VEL
LIN {X 0,Y 74.247,Z 472.067,A -85,B 0,C 180,E1 -30065.505,E2 -30065.505} C_VEL
LIN {X 0,Y 68.867,Z 473.249,A -85,B 0,C 180,E1 -30067.254,E2 -30067.254} C_VEL
LIN {X 0,Y 59.305,Z 474.623,A -85,B 0,C 180,E1 -30069.279,E2 -30069.279} C_VEL
LIN {X 0,Y 49.784,Z 475.225,A -85,B 0,C 180,E1 -30072.1,E2 -30072.1} C_VEL
LIN {X 0,Y 44.637,Z 475.161,A -85,B 0,C 180,E1 -30075.612,E2 -30075.612} C_VEL
LIN {X 0,Y 38.277,Z 474.667,A -85,B 0,C 180,E1 -30083.352,E2 -30083.352} C_VEL
LIN {X 0,Y 33.334,Z 473.7,A -85,B 0,C 180,E1 -30092.499,E2 -30092.499} C_VEL
LIN {X 0,Y 28.963,Z 472.042,A -85,B 0,C 180,E1 -30106.621,E2 -30106.621} C_VEL
LIN {X 0,Y 26.573,Z 469.345,A -85,B 0,C 180,E1 -30126.621,E2 -30126.621} C_VEL
LIN {X 0,Y 28.114,Z 464.688,A -85,B 0,C 180,E1 -30152.841,E2 -30152.841} C_VEL
LIN {X 0,Y 33.156,Z 459.065,A -85,B 0,C 180,E1 -30171.77,E2 -30171.77} C_VEL
LIN {X 0,Y 40.024,Z 452.261,A -85,B 0,C 180,E1 -30184.793,E2 -30184.793} C_VEL
LIN {X 0,Y 48.211,Z 443.81,A -85,B 0,C 180,E1 -30193.819,E2 -30193.819} C_VEL
LIN {X 0,Y 55.637,Z 435.096,A -85,B 0,C 180,E1 -30199.277,E2 -30199.277} C_VEL
LIN {X 0,Y 62.665,Z 425.505,A -85,B 0,C 180,E1 -30203.039,E2 -30203.039} C_VEL
LIN {X 0,Y 69.898,Z 413.581,A -85,B 0,C 180,E1 -30206.045,E2 -30206.045} C_VEL
LIN {X 0,Y 75.559,Z 401.655,A -85,B 0,C 180,E1 -30208.072,E2 -30208.072} C_VEL
LIN {X 0,Y 80.081,Z 389.217,A -85,B 0,C 180,E1 -30209.443,E2 -30209.443} C_VEL
LIN {X 0,Y 83.373,Z 376.515,A -85,B 0,C 180,E1 -30210.361,E2 -30210.361} C_VEL
LIN {X 0,Y 85.418,Z 363.546,A -85,B 0,C 180,E1 -30210.895,E2 -30210.895} C_VEL
LIN {X 0,Y 87.073,Z 349.233,A -85,B 0,C 180,E1 -30211.414,E2 -30211.414} C_VEL
LIN {X 0,Y 85.762,Z 344.902,A -85,B 0,C 180,E1 -30215.461,E2 -30215.461} C_VEL
LIN {X 0,Y 84.578,Z 341.248,A -85,B 0,C 180,E1 -30220.433,E2 -30220.433} C_VEL
LIN {X 0,Y 83.762,Z 337.994,A -85,B 0,C 180,E1 -30227.701,E2 -30227.701} C_VEL
LIN {X 0,Y 83.89,Z 337.976,A -85,B 0,C 180,E1 -30235.468,E2 -30235.468} C_VEL
LIN {X 0,Y 84.619,Z 341.148,A -85,B 0,C 180,E1 -30241.509,E2 -30241.509} C_VEL
LIN {X 0,Y 85.677,Z 344.588,A -85,B 0,C 180,E1 -30246.054,E2 -30246.054} C_VEL
LIN {X 0,Y 87.108,Z 349.408,A -85,B 0,C 180,E1 -30250.526,E2 -30250.526} C_VEL
LIN {X 0,Y 84.015,Z 373.917,A -85,B 0,C 180,E1 -30251.511,E2 -30251.511} C_VEL
LIN {X 0,Y 80.921,Z 387.058,A -85,B 0,C 180,E1 -30252.236,E2 -30252.236} C_VEL
LIN {X 0,Y 76.805,Z 399.379,A -85,B 0,C 180,E1 -30253.543,E2 -30253.543} C_VEL
LIN {X 0,Y 71.858,Z 410.353,A -85,B 0,C 180,E1 -30255.033,E2 -30255.033} C_VEL
LIN {X 0,Y 67.758,Z 417.864,A -85,B 0,C 180,E1 -30256.386,E2 -30256.386} C_VEL
LIN {X 0,Y 61.401,Z 427.941,A -85,B 0,C 180,E1 -30259.22,E2 -30259.22} C_VEL
LIN {X 0,Y 55.457,Z 435.882,A -85,B 0,C 180,E1 -30262.429,E2 -30262.429} C_VEL
LIN {X 0,Y 47.812,Z 444.842,A -85,B 0,C 180,E1 -30268.127,E2 -30268.127} C_VEL
LIN {X 0,Y 39.679,Z 453.193,A -85,B 0,C 180,E1 -30277.158,E2 -30277.158} C_VEL
LIN {X 0,Y 32.908,Z 459.894,A -85,B 0,C 180,E1 -30290.162,E2 -30290.162} C_VEL
LIN {X 0,Y 28.426,Z 465.21,A -85,B 0,C 180,E1 -30308.237,E2 -30308.237} C_VEL
LIN {X 0,Y 27.129,Z 469.306,A -85,B 0,C 180,E1 -30330.005,E2 -30330.005} C_VEL
LIN {X 0,Y 27.731,Z 471.407,A -85,B 0,C 180,E1 -30344.686,E2 -30344.686} C_VEL
LIN {X 0,Y 33.201,Z 474.293,A -85,B 0,C 180,E1 -30369.428,E2 -30369.428} C_VEL
LIN {X 0,Y 42.666,Z 475.643,A -85,B 0,C 180,E1 -30385.453,E2 -30385.453} C_VEL
LIN {X 0,Y 54.318,Z 475.425,A -85,B 0,C 180,E1 -30394.924,E2 -30394.924} C_VEL
LIN {X 0,Y 66.95,Z 473.716,A -85,B 0,C 180,E1 -30400.872,E2 -30400.872} C_VEL
LIN {X 0,Y 75.577,Z 471.681,A -85,B 0,C 180,E1 -30403.777,E2 -30403.777} C_VEL
LIN {X 0,Y 86.719,Z 468.077,A -85,B 0,C 180,E1 -30406.541,E2 -30406.541} C_VEL
LIN {X 0,Y 96.853,Z 463.751,A -85,B 0,C 180,E1 -30408.416,E2 -30408.416} C_VEL
LIN {X 0,Y 107.102,Z 458.264,A -85,B 0,C 180,E1 -30409.838,E2 -30409.838} C_VEL
LIN {X 0,Y 115.774,Z 452.599,A -85,B 0,C 180,E1 -30410.857,E2 -30410.857} C_VEL
LIN {X 0,Y 117.415,Z 451.422,A -85,B 0,C 180,E1 -30411.604,E2 -30411.604} C_VEL
LIN {X 0,Y 106.214,Z 458.715,A -85,B 0,C 180,E1 -30412.997,E2 -30412.997} C_VEL
LIN {X 0,Y 95.29,Z 464.369,A -85,B 0,C 180,E1 -30414.684,E2 -30414.684} C_VEL
LIN {X 0,Y 84.467,Z 468.723,A -85,B 0,C 180,E1 -30416.837,E2 -30416.837} C_VEL
LIN {X 0,Y 72.786,Z 472.165,A -85,B 0,C 180,E1 -30419.975,E2 -30419.975} C_VEL
LIN {X 0,Y 63.37,Z 474.006,A -85,B 0,C 180,E1 -30423.473,E2 -30423.473} C_VEL
LIN {X 0,Y 55.834,Z 474.896,A -85,B 0,C 180,E1 -30427.198,E2 -30427.198} C_VEL
LIN {X 0,Y 44.637,Z 475.161,A -85,B 0,C 180,E1 -30435.612,E2 -30435.612} C_VEL
LIN {X 0,Y 39.696,Z 474.932,A -85,B 0,C 180,E1 -30440.004,E2 -30440.004} C_VEL
LIN {X 0,Y 31.004,Z 473.807,A -85,B 0,C 180,E1 -30447.584,E2 -30447.584} C_VEL
LIN {X 0,Y 24.568,Z 472.302,A -85,B 0,C 180,E1 -30456.882,E2 -30456.882} C_VEL
LIN {X 0,Y 21.041,Z 470.871,A -85,B 0,C 180,E1 -30468.395,E2 -30468.395} C_VEL
LIN {X 0,Y 20.333,Z 470.313,A -85,B 0,C 180,E1 -30473.3,E2 -30473.3} C_VEL
LIN {X 0,Y 19.563,Z 467.336,A -85,B 0,C 180,E1 -30499.645,E2 -30499.645} C_VEL
LIN {X 0,Y 23.327,Z 462.646,A -85,B 0,C 180,E1 -30527.528,E2 -30527.528} C_VEL
LIN {X 0,Y 30.247,Z 456.694,A -85,B 0,C 180,E1 -30545.508,E2 -30545.508} C_VEL
LIN {X 0,Y 38.739,Z 449.259,A -85,B 0,C 180,E1 -30556.519,E2 -30556.519} C_VEL
LIN {X 0,Y 47.372,Z 440.679,A -85,B 0,C 180,E1 -30563.301,E2 -30563.301} C_VEL
LIN {X 0,Y 55.278,Z 431.521,A -85,B 0,C 180,E1 -30567.379,E2 -30567.379} C_VEL
LIN {X 0,Y 62.798,Z 421.037,A -85,B 0,C 180,E1 -30570.145,E2 -30570.145} C_VEL
LIN {X 0,Y 69.518,Z 409.417,A -85,B 0,C 180,E1 -30572.197,E2 -30572.197} C_VEL
LIN {X 0,Y 74.992,Z 397.259,A -85,B 0,C 180,E1 -30573.653,E2 -30573.653} C_VEL
LIN {X 0,Y 79.418,Z 383.758,A -85,B 0,C 180,E1 -30574.712,E2 -30574.712} C_VEL
LIN {X 0,Y 82.185,Z 371.37,A -85,B 0,C 180,E1 -30575.252,E2 -30575.252} C_VEL
LIN {X 0,Y 84.576,Z 352.659,A -85,B 0,C 180,E1 -30575.878,E2 -30575.878} C_VEL
LIN {X 0,Y 83.593,Z 348.986,A -85,B 0,C 180,E1 -30580.373,E2 -30580.373} C_VEL
LIN {X 0,Y 83.111,Z 347.312,A -85,B 0,C 180,E1 -30583.519,E2 -30583.519} C_VEL
LIN {X 0,Y 82.815,Z 344.911,A -85,B 0,C 180,E1 -30588.8,E2 -30588.8} C_VEL
LIN {X 0,Y 82.903,Z 344.933,A -85,B 0,C 180,E1 -30594.413,E2 -30594.413} C_VEL
LIN {X 0,Y 83.391,Z 347.815,A -85,B 0,C 180,E1 -30600.022,E2 -30600.022} C_VEL
LIN {X 0,Y 84.3,Z 351.5,A -85,B 0,C 180,E1 -30604.804,E2 -30604.804} C_VEL
LIN {X 0,Y 84.614,Z 352.86,A -85,B 0,C 180,E1 -30606.118,E2 -30606.118} C_VEL
LIN {X 0,Y 81.924,Z 373.389,A -85,B 0,C 180,E1 -30606.846,E2 -30606.846} C_VEL
LIN {X 0,Y 78.799,Z 386.48,A -85,B 0,C 180,E1 -30607.373,E2 -30607.373} C_VEL
LIN {X 0,Y 74.599,Z 398.839,A -85,B 0,C 180,E1 -30608.44,E2 -30608.44} C_VEL
LIN {X 0,Y 69.495,Z 409.904,A -85,B 0,C 180,E1 -30609.609,E2 -30609.609} C_VEL
LIN {X 0,Y 65.254,Z 417.448,A -85,B 0,C 180,E1 -30610.66,E2 -30610.66} C_VEL
LIN {X 0,Y 58.6,Z 427.593,A -85,B 0,C 180,E1 -30612.994,E2 -30612.994} C_VEL
LIN {X 0,Y 52.902,Z 434.891,A -85,B 0,C 180,E1 -30615.443,E2 -30615.443} C_VEL
LIN {X 0,Y 46.459,Z 442.134,A -85,B 0,C 180,E1 -30619.022,E2 -30619.022} C_VEL
LIN {X 0,Y 37.295,Z 451.061,A -85,B 0,C 180,E1 -30626.486,E2 -30626.486} C_VEL
LIN {X 0,Y 29.007,Z 458.151,A -85,B 0,C 180,E1 -30638.061,E2 -30638.061} C_VEL
LIN {X 0,Y 23.568,Z 462.969,A -85,B 0,C 180,E1 -30653.395,E2 -30653.395} C_VEL
LIN {X 0,Y 20.158,Z 467.577,A -85,B 0,C 180,E1 -30679.968,E2 -30679.968} C_VEL
LIN {X 0,Y 20.251,Z 469.973,A -85,B 0,C 180,E1 -30699.999,E2 -30699.999} C_VEL
LIN {X 0,Y 23.767,Z 472.724,A -85,B 0,C 180,E1 -30726.264,E2 -30726.264} C_VEL
LIN {X 0,Y 33.266,Z 474.936,A -85,B 0,C 180,E1 -30747.686,E2 -30747.686} C_VEL
LIN {X 0,Y 45.285,Z 475.645,A -85,B 0,C 180,E1 -30758.625,E2 -30758.625} C_VEL
LIN {X 0,Y 58.281,Z 474.782,A -85,B 0,C 180,E1 -30764.739,E2 -30764.739} C_VEL
LIN {X 0,Y 71.705,Z 472.417,A -85,B 0,C 180,E1 -30768.565,E2 -30768.565} C_VEL
LIN {X 0,Y 81.921,Z 469.545,A -85,B 0,C 180,E1 -30770.614,E2 -30770.614} C_VEL
LIN {X 0,Y 85.346,Z 468.36,A -85,B 0,C 180,E1 -30771.184,E2 -30771.184} C_VEL
LIN {X 0,Y 85.224,Z 468.393,A -85,B 0,C 180,E1 -30771.73,E2 -30771.73} C_VEL
LIN {X 0,Y 77.886,Z 470.744,A -85,B 0,C 180,E1 -30773.026,E2 -30773.026} C_VEL
LIN {X 0,Y 70.595,Z 472.559,A -85,B 0,C 180,E1 -30774.603,E2 -30774.603} C_VEL
LIN {X 0,Y 63.369,Z 473.913,A -85,B 0,C 180,E1 -30776.54,E2 -30776.54} C_VEL
LIN {X 0,Y 53.912,Z 475.019,A -85,B 0,C 180,E1 -30779.966,E2 -30779.966} C_VEL
LIN {X 0,Y 42.43,Z 475.289,A -85,B 0,C 180,E1 -30786.347,E2 -30786.347} C_VEL
LIN {X 0,Y 35.944,Z 474.875,A -85,B 0,C 180,E1 -30792.122,E2 -30792.122} C_VEL
LIN {X 0,Y 29.939,Z 474.003,A -85,B 0,C 180,E1 -30800.105,E2 -30800.105} C_VEL
LIN {X 0,Y 23.157,Z 472.073,A -85,B 0,C 180,E1 -30817.271,E2 -30817.271} C_VEL
LIN {X 0,Y 20.333,Z 470.313,A -85,B 0,C 180,E1 -30833.3,E2 -30833.3} C_VEL
LIN {X 0,Y 18.716,Z 468.557,A -85,B 0,C 180,E1 -30849.153,E2 -30849.153} C_VEL
LIN {X 0,Y 17.64,Z 466.54,A -85,B 0,C 180,E1 -30866.511,E2 -30866.511} C_VEL
LIN {X 0,Y 20.444,Z 460.825,A -85,B 0,C 180,E1 -30904.882,E2 -30904.882} C_VEL
LIN {X 0,Y 24.176,Z 457.887,A -85,B 0,C 180,E1 -30914.413,E2 -30914.413} C_VEL
LIN {X 0,Y 32.556,Z 451.576,A -85,B 0,C 180,E1 -30924.042,E2 -30924.042} C_VEL
LIN {X 0,Y 40.777,Z 444.466,A -85,B 0,C 180,E1 -30929.508,E2 -30929.508} C_VEL
LIN {X 0,Y 49.219,Z 435.882,A -85,B 0,C 180,E1 -30933.176,E2 -30933.176} C_VEL
LIN {X 0,Y 56.955,Z 426.417,A -85,B 0,C 180,E1 -30935.505,E2 -30935.505} C_VEL
LIN {X 0,Y 64.745,Z 414.647,A -85,B 0,C 180,E1 -30937.313,E2 -30937.313} C_VEL
LIN {X 0,Y 70.791,Z 403.049,A -85,B 0,C 180,E1 -30938.544,E2 -30938.544} C_VEL
LIN {X 0,Y 75.621,Z 390.838,A -85,B 0,C 180,E1 -30939.359,E2 -30939.359} C_VEL
